// TIA Portal project "chiller" (V19)

(* hardware
DEVICE "S7-1500/ET200MP station_1"  S7-1500 station
   slot 0: "Rail_0"  Rack  6ES7 590-1***0-0AA0
   slot 1: "PLC_1"  CPU 1513-1 PN  6ES7 513-1AM03-0AB0  V3.1
      slot 3: "CPU display_1"  6ES7591-1AA00-0AA0
      slot 32768: "PROFINET interface_1"  X1
         slot 32769: "Port_1"  X1 P1
         slot 32770: "Port_2"  X1 P2
      slot 34817: "Virtual CP interface port_1"  Virtual CP interface port  Virtual CP interface port
   slot 2: "DI 16x24VDC BA_1"  DI 16x24VDC BA  6ES7 521-1BH10-0AA0  V1.1
   slot 3: "DI 16x24VDC BA_2"  DI 16x24VDC BA  6ES7 521-1BH10-0AA0  V1.1
   slot 4: "DQ 16x24VDC/0.5A BA_1"  DQ 16x24VDC/0.5A BA  6ES7 522-1BH10-0AA0  V1.1
   slot 5: "AI 16xI BA_1"  AI 16xI BA  6ES7 531-7MH00-0AB0  V1.0
   slot 6: "AQ 8xU/I HS_1"  AQ 8xU/I HS  6ES7 532-5HF00-0AB0  V2.2
DEVICE "HMI_1"  TP700 Comfort
   slot 0: "HMI_1"  TP700 Comfort  6AV2 124-0GC01-0AX0  17.0.0.0
   slot 1: "HMI_RT_1"  TP700 Comfort  6AV2 124-0GC01-0AX0  17.0.0.0
   slot 5: "HMI_1.IE_CP_1"  PROFINET Interface  17.0.0.0
      slot 1: "PROFINET Interface_1"  PROFINET Interface
         slot 1: "Port_1"  Port
         slot 2: "Port_2"  Port
   slot 7: "HMI_1.MPI/DP_CP_1"  MPI/DP Interface  17.0.0.0
*)

// ===== PLC "PLC_1"  CPU 1513-1 PN =====

VAR_GLOBAL   // PLC tag table "IO_Inputs"
   "I0.0" AT %I0.0 : Bool;
   "I0.1" AT %I0.1 : Bool;
   "I0.2" AT %I0.2 : Bool;
   "I0.3" AT %I0.3 : Bool;
   "I0.4" AT %I0.4 : Bool;
   "I0.5" AT %I0.5 : Bool;
   "I0.6" AT %I0.6 : Bool;
   "I0.7" AT %I0.7 : Bool;
   "I1.0" AT %I1.0 : Bool;
   "I1.1" AT %I1.1 : Bool;
   "I1.2" AT %I1.2 : Bool;
   "I1.3" AT %I1.3 : Bool;
   "I1.4" AT %I1.4 : Bool;
   "I1.5" AT %I1.5 : Bool;
   "I1.6" AT %I1.6 : Bool;
   "I1.7" AT %I1.7 : Bool;
   "I_Comp06_OffFb" AT %I2.0 : Bool;
   "I_Comp06_Fault" AT %I2.1 : Bool;
   "I_Comp07_OnFb" AT %I2.2 : Bool;
   "I_Comp07_OffFb" AT %I2.3 : Bool;
   "I_Comp07_Fault" AT %I2.4 : Bool;
   "I_Comp08_OnFb" AT %I2.5 : Bool;
   "I_Comp08_OffFb" AT %I2.6 : Bool;
   "I_Comp08_Fault" AT %I2.7 : Bool;
   "System_Byte" AT %MB1 : Byte;
   "FirstScan" AT %M1.0 : Bool;
   "DiagStatusUpdate" AT %M1.1 : Bool;
   "AlwaysTRUE" AT %M1.2 : Bool;
   "AlwaysFALSE" AT %M1.3 : Bool;
   "Clock_Byte" AT %MB10 : Byte;
   "Clock_10Hz" AT %M10.0 : Bool;
   "Clock_5Hz" AT %M10.1 : Bool;
   "Clock_2.5Hz" AT %M10.2 : Bool;
   "Clock_2Hz" AT %M10.3 : Bool;
   "Clock_1.25Hz" AT %M10.4 : Bool;
   "Clock_1Hz" AT %M10.5 : Bool;
   "Clock_0.625Hz" AT %M10.6 : Bool;
   "Clock_0.5Hz" AT %M10.7 : Bool;
   "Tag_1" AT %I34.0 : Bool;
END_VAR

VAR_GLOBAL   // PLC tag table "IO_Outputs"
   "Q_Comp01_Start" AT %I3.0 : Bool;
   "Q_Comp02_Start" AT %I3.1 : Bool;
   "Q_Comp03_Start" AT %I3.2 : Bool;
   "Q_Comp04_Start" AT %I3.3 : Bool;
   "Q_Comp05_Start" AT %I3.4 : Bool;
   "Q_Comp06_Start" AT %I3.5 : Bool;
   "Q_Comp07_Start" AT %I3.6 : Bool;
   "Q_Comp08_Start" AT %I3.7 : Bool;
END_VAR

TYPE "UDT_Process"
   STRUCT
      WaterOutletTemp : Real;
      WaterTempSetPoint : Real;
      GasPressure : Real;
      GasPressureSetPoint : Real;
      CompressorDemand : Real;
      FanDemand : Real;
      RunningCompressorCount : Int;
      RunningFanCount : Int;
      CompressorPercent : Real;
      FanPercent : Real;
      RequiredCompressorCount : Int;
      RequestedCompressorCount : Int;
      RequiredFanCount : Int;
      RequestedFanCount : Int;
   END_STRUCT;
END_TYPE

TYPE "UDT_Fan"
   STRUCT
      IO : Struct
         DI_OnFeedback : Bool;
         DI_OffFeedback : Bool;
         DI_Fault : Bool;
         DO_Start : Bool;
      END_STRUCT;
      Cfg : Struct
         Enabled : Bool;
      END_STRUCT;
      Sts : Struct
         Runnig : Bool;
         Ready : Bool;
         Status : Int;
      END_STRUCT;
      Cmd : Struct
         StartRequest : Bool;
         ResetFault : Bool;
      END_STRUCT;
      Flt : Struct
         FeedbackFault : Bool;
         AnyFault : Bool;
      END_STRUCT;
   END_STRUCT;
END_TYPE

TYPE "UDT_Compressor"
   STRUCT
      Cfg : Struct
         Enabled : Bool;
      END_STRUCT;
      Sts : Struct
         Running : Bool;
         Ready : Bool;
         Status : Int;
         RunSeconds : DInt;
         RunHours : Real;
      END_STRUCT;
      Cmd : Struct
         StartRequest : Bool;
         ResetFault : Bool;
         ResetRuntime : Bool;
      END_STRUCT;
      Flt : Struct
         FeedbackFault : Bool;
         AnyFault : Bool;
      END_STRUCT;
      IO : Struct
         DI_OnFeedback : Bool;
         DI_OffFeedback : Bool;
         DI_Fault : Bool;
         DO_Start : Bool;
      END_STRUCT;
   END_STRUCT;
END_TYPE

TYPE "UDT_TimingParams"
   STRUCT
      MinOffTime : Time;
      MinOnTime : Time;
      FeedbackTime : Time;
   END_STRUCT;
END_TYPE

// folder: 00_main

DATA_BLOCK "DB_EquipmentMain"   // DB3
{ S7_Optimized_Access := 'TRUE' }
VERSION : 0.1
// stored: InstanceOfName FB_EquipmentMain
"FB_EquipmentMain"
BEGIN
END_DATA_BLOCK

DATA_BLOCK "DB_MachineMain"   // DB5
{ S7_Optimized_Access := 'TRUE' }
VERSION : 0.1
// stored: InstanceOfName FB_MachineMain
"FB_MachineMain"
BEGIN
END_DATA_BLOCK

DATA_BLOCK "DB_SimulationMain"   // DB6
{ S7_Optimized_Access := 'TRUE' }
VERSION : 0.1
// stored: InstanceOfName FB_SimulationMain
"FB_SimulationMain"
BEGIN
END_DATA_BLOCK

// folder: 03_globalData

DATA_BLOCK "Db_Equipment"   // DB1
{ S7_Optimized_Access := 'TRUE' }
VERSION : 0.1
   VAR
      Compressor : Array[1..8] of "UDT_Compressor";
      Process : "UDT_Process";
      Fan : Array[1..12] of "UDT_Fan";
      CompressorTiming : "UDT_TimingParams";
      FanTiming : "UDT_TimingParams";
   END_VAR
BEGIN
END_DATA_BLOCK

DATA_BLOCK "DB_Machine"   // DB2
{ S7_Optimized_Access := 'TRUE' }
VERSION : 0.1
   VAR
      AutoMode : Bool;
      ManualMode : Bool;
      StartRequest : Bool;
      StopRequest : Bool;
      Running : Bool;
      Ready : Bool;
      AnyFault : Bool;
      DisableAllEquipment : Bool;
      EnableAllEquipment : Bool;
      ResetAllEquipmentFaults : Bool;
      WaterFlowOK : Bool;
      LowTempFault : Bool;
      LowTempLimit : Real;
      WaterFlowFaultDelay : Time;
      LowTempFaultDelay : Time;
      WaterFlowFault : Bool;
   END_VAR
BEGIN
END_DATA_BLOCK

DATA_BLOCK "DB_Simulation"   // DB4
{ S7_Optimized_Access := 'TRUE' }
VERSION : 0.1
   VAR
      Enabled : Bool;
      CompressorOnFb : Array[1..8] of Bool;
      CompressorOffFb : Array[1..8] of Bool;
      CompressorFault : Array[1..8] of Bool;
      FanOnFb : Array[1..12] of Bool;
      FanOffFb : Array[1..12] of Bool;
      FanFaultFb : Array[1..12] of Bool;
   END_VAR
BEGIN
END_DATA_BLOCK

DATA_BLOCK "DB_Alarm"   // DB9
{ S7_Optimized_Access := 'TRUE' }
VERSION : 0.1
   VAR
      AlarmWord1 : Word;
      AlarmWord2 : Word;
   END_VAR
BEGIN
END_DATA_BLOCK

// folder: 00_main

FUNCTION_BLOCK "FB_MachineMain"   // FB5, LAD
{ S7_Optimized_Access := 'TRUE' }
VERSION : 0.1
   VAR
      tWaterFlowFault : TON_TIME;
      tLowTempFault : TON_TIME;
   END_VAR
   VAR_TEMP
      WaterFlowTimeout : Bool;
      LowTempTimeout : Bool;
   END_VAR
BEGIN

REGION Network 1
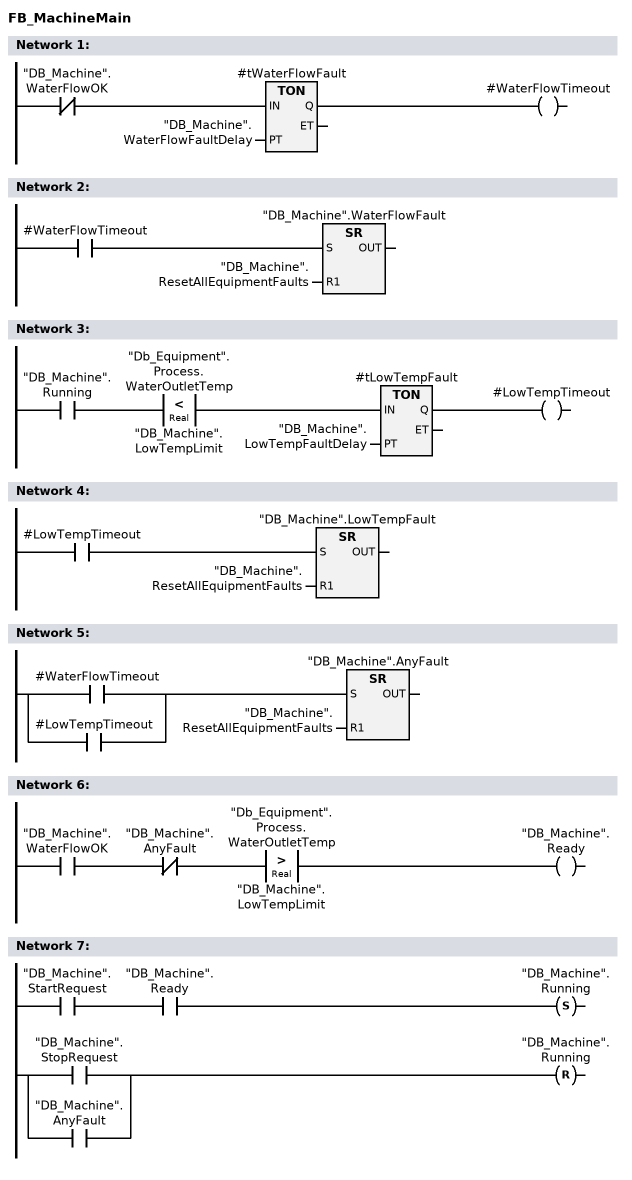
   #tWaterFlowFault(IN := NOT "DB_Machine".WaterFlowOK, PT := "DB_Machine".WaterFlowFaultDelay);   // TON
   #WaterFlowTimeout := #tWaterFlowFault.Q;
END_REGION

REGION Network 2
   RUNG wire#powerrail
      Contact( #WaterFlowTimeout )
      S_SR(operand := "DB_Machine".WaterFlowFault, r1 := "DB_Machine".ResetAllEquipmentFaults)
   END_RUNG
   // the same network as SCL:
   IF #WaterFlowTimeout THEN
       "DB_Machine".WaterFlowFault := TRUE;   // SR flip-flop
   END_IF;
   IF "DB_Machine".ResetAllEquipmentFaults THEN "DB_Machine".WaterFlowFault := FALSE; END_IF;
END_REGION

REGION Network 3
   #tLowTempFault(IN := "DB_Machine".Running AND ("Db_Equipment".Process.WaterOutletTemp < "DB_Machine".LowTempLimit),   // TON
                  PT := "DB_Machine".LowTempFaultDelay);
   #LowTempTimeout := #tLowTempFault.Q;
END_REGION

REGION Network 4
   RUNG wire#powerrail
      Contact( #LowTempTimeout )
      S_SR(operand := "DB_Machine".LowTempFault, r1 := "DB_Machine".ResetAllEquipmentFaults)
   END_RUNG
   // the same network as SCL:
   IF #LowTempTimeout THEN
       "DB_Machine".LowTempFault := TRUE;   // SR flip-flop
   END_IF;
   IF "DB_Machine".ResetAllEquipmentFaults THEN "DB_Machine".LowTempFault := FALSE; END_IF;
END_REGION

REGION Network 5
   RUNG wire#powerrail
      Contact( #WaterFlowTimeout )
      wire#w1
      S_SR(operand := "DB_Machine".AnyFault, r1 := "DB_Machine".ResetAllEquipmentFaults)
   END_RUNG
   RUNG wire#powerrail
      Contact( #LowTempTimeout )
   END_RUNG wire#w1
   // the same network as SCL:
   IF #WaterFlowTimeout OR #LowTempTimeout THEN
       "DB_Machine".AnyFault := TRUE;   // SR flip-flop
   END_IF;
   IF "DB_Machine".ResetAllEquipmentFaults THEN "DB_Machine".AnyFault := FALSE; END_IF;
END_REGION

REGION Network 6
   RUNG wire#powerrail
      Contact( "DB_Machine".WaterFlowOK )
      I_Contact( "DB_Machine".AnyFault )
      { S7_Templates := "SrcType := Real" } GT_Contact(in1 := "Db_Equipment".Process.WaterOutletTemp, in2 := "DB_Machine".LowTempLimit)
      Coil( "DB_Machine".Ready )
   END_RUNG
   // the same network as SCL:
   "DB_Machine".Ready := "DB_Machine".WaterFlowOK AND NOT "DB_Machine".AnyFault AND ("Db_Equipment".Process.WaterOutletTemp > "DB_Machine".LowTempLimit);
END_REGION

REGION Network 7
   RUNG wire#powerrail
      Contact( "DB_Machine".StartRequest )
      Contact( "DB_Machine".Ready )
      S_Coil( "DB_Machine".Running )
   END_RUNG
   RUNG wire#powerrail
      Contact( "DB_Machine".StopRequest )
      wire#w1
      R_Coil( "DB_Machine".Running )
   END_RUNG
   RUNG wire#powerrail
      Contact( "DB_Machine".AnyFault )
   END_RUNG wire#w1
   // the same network as SCL:
   IF "DB_Machine".StartRequest AND "DB_Machine".Ready THEN "DB_Machine".Running := TRUE; END_IF;
   IF "DB_Machine".StopRequest OR "DB_Machine".AnyFault THEN "DB_Machine".Running := FALSE; END_IF;
END_REGION
END_FUNCTION_BLOCK

FUNCTION_BLOCK "FB_EquipmentMain"   // FB6, LAD
{ S7_Optimized_Access := 'TRUE' }
VERSION : 0.1
   VAR
      Comp01 : "FB_Compressor";
      Comp02 : "FB_Compressor";
      Comp03 : "FB_Compressor";
      Comp04 : "FB_Compressor";
      Comp05 : "FB_Compressor";
      Comp06 : "FB_Compressor";
      Comp07 : "FB_Compressor";
      Comp08 : "FB_Compressor";
      Comp09 : "FB_Compressor";
      FB_CompressorManager : "FB_CompressorManager";
      Fan01 : "FB_Fan";
      Fan02 : "FB_Fan";
      Fan03 : "FB_Fan";
      Fan04 : "FB_Fan";
      Fan05 : "FB_Fan";
      Fan06 : "FB_Fan";
      Fan07 : "FB_Fan";
      Fan08 : "FB_Fan";
      Fan09 : "FB_Fan";
      Fan10 : "FB_Fan";
      Fan11 : "FB_Fan";
      Fan12 : "FB_Fan";
      FanManager : "FB_FanManager";
   END_VAR
   VAR_TEMP
      FanControlEnable : Bool;
   END_VAR
BEGIN

REGION Network 1
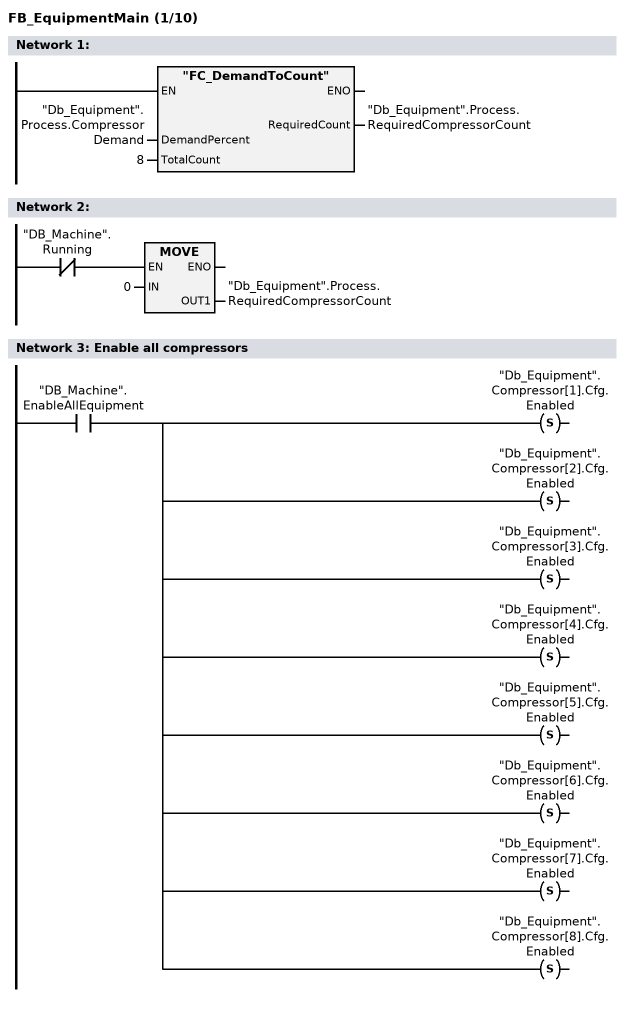
   RUNG wire#powerrail
      "FC_DemandToCount"(DemandPercent := "Db_Equipment".Process.CompressorDemand, TotalCount := 8, RequiredCount => "Db_Equipment".Process.RequiredCompressorCount)
   END_RUNG
   // the same network as SCL:
   "FC_DemandToCount"(DemandPercent := "Db_Equipment".Process.CompressorDemand,
                      TotalCount := 8,
                      RequiredCount => "Db_Equipment".Process.RequiredCompressorCount);
END_REGION

REGION Network 2
   RUNG wire#powerrail
      I_Contact( "DB_Machine".Running )
      Move(in := 0, out1 => "Db_Equipment".Process.RequiredCompressorCount)
   END_RUNG
   // the same network as SCL:
   IF NOT "DB_Machine".Running THEN "Db_Equipment".Process.RequiredCompressorCount := 0; END_IF;
END_REGION

REGION Network 3: Enable all compressors
   RUNG wire#powerrail
      Contact( "DB_Machine".EnableAllEquipment )
      wire#w1
      S_Coil( "Db_Equipment".Compressor[1].Cfg.Enabled )
   END_RUNG
   RUNG wire#w1
      S_Coil( "Db_Equipment".Compressor[2].Cfg.Enabled )
   END_RUNG
   RUNG wire#w1
      S_Coil( "Db_Equipment".Compressor[3].Cfg.Enabled )
   END_RUNG
   RUNG wire#w1
      S_Coil( "Db_Equipment".Compressor[4].Cfg.Enabled )
   END_RUNG
   RUNG wire#w1
      S_Coil( "Db_Equipment".Compressor[5].Cfg.Enabled )
   END_RUNG
   RUNG wire#w1
      S_Coil( "Db_Equipment".Compressor[6].Cfg.Enabled )
   END_RUNG
   RUNG wire#w1
      S_Coil( "Db_Equipment".Compressor[7].Cfg.Enabled )
   END_RUNG
   RUNG wire#w1
      S_Coil( "Db_Equipment".Compressor[8].Cfg.Enabled )
   END_RUNG
   // the same network as SCL:
   IF "DB_Machine".EnableAllEquipment THEN
       "Db_Equipment".Compressor[1].Cfg.Enabled := TRUE;
       "Db_Equipment".Compressor[2].Cfg.Enabled := TRUE;
       "Db_Equipment".Compressor[3].Cfg.Enabled := TRUE;
       "Db_Equipment".Compressor[4].Cfg.Enabled := TRUE;
       "Db_Equipment".Compressor[5].Cfg.Enabled := TRUE;
       "Db_Equipment".Compressor[6].Cfg.Enabled := TRUE;
       "Db_Equipment".Compressor[7].Cfg.Enabled := TRUE;
       "Db_Equipment".Compressor[8].Cfg.Enabled := TRUE;
   END_IF;
END_REGION

REGION Network 4: Enable all fans
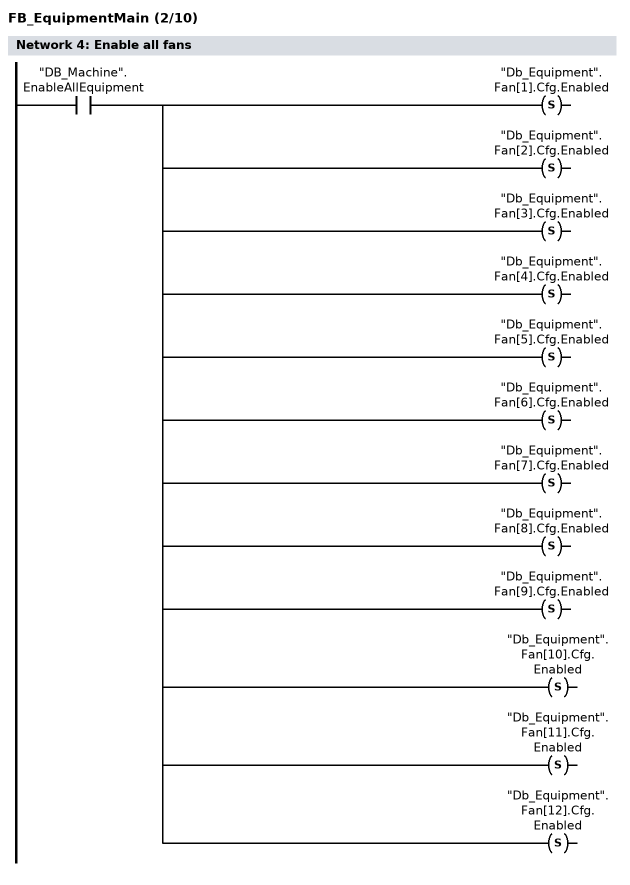
   RUNG wire#powerrail
      Contact( "DB_Machine".EnableAllEquipment )
      wire#w1
      S_Coil( "Db_Equipment".Fan[1].Cfg.Enabled )
   END_RUNG
   RUNG wire#w1
      S_Coil( "Db_Equipment".Fan[2].Cfg.Enabled )
   END_RUNG
   RUNG wire#w1
      S_Coil( "Db_Equipment".Fan[3].Cfg.Enabled )
   END_RUNG
   RUNG wire#w1
      S_Coil( "Db_Equipment".Fan[4].Cfg.Enabled )
   END_RUNG
   RUNG wire#w1
      S_Coil( "Db_Equipment".Fan[5].Cfg.Enabled )
   END_RUNG
   RUNG wire#w1
      S_Coil( "Db_Equipment".Fan[6].Cfg.Enabled )
   END_RUNG
   RUNG wire#w1
      S_Coil( "Db_Equipment".Fan[7].Cfg.Enabled )
   END_RUNG
   RUNG wire#w1
      S_Coil( "Db_Equipment".Fan[8].Cfg.Enabled )
   END_RUNG
   RUNG wire#w1
      S_Coil( "Db_Equipment".Fan[9].Cfg.Enabled )
   END_RUNG
   RUNG wire#w1
      S_Coil( "Db_Equipment".Fan[10].Cfg.Enabled )
   END_RUNG
   RUNG wire#w1
      S_Coil( "Db_Equipment".Fan[11].Cfg.Enabled )
   END_RUNG
   RUNG wire#w1
      S_Coil( "Db_Equipment".Fan[12].Cfg.Enabled )
   END_RUNG
   // the same network as SCL:
   IF "DB_Machine".EnableAllEquipment THEN
       "Db_Equipment".Fan[1].Cfg.Enabled := TRUE;
       "Db_Equipment".Fan[2].Cfg.Enabled := TRUE;
       "Db_Equipment".Fan[3].Cfg.Enabled := TRUE;
       "Db_Equipment".Fan[4].Cfg.Enabled := TRUE;
       "Db_Equipment".Fan[5].Cfg.Enabled := TRUE;
       "Db_Equipment".Fan[6].Cfg.Enabled := TRUE;
       "Db_Equipment".Fan[7].Cfg.Enabled := TRUE;
       "Db_Equipment".Fan[8].Cfg.Enabled := TRUE;
       "Db_Equipment".Fan[9].Cfg.Enabled := TRUE;
       "Db_Equipment".Fan[10].Cfg.Enabled := TRUE;
       "Db_Equipment".Fan[11].Cfg.Enabled := TRUE;
       "Db_Equipment".Fan[12].Cfg.Enabled := TRUE;
   END_IF;
END_REGION

REGION Network 5
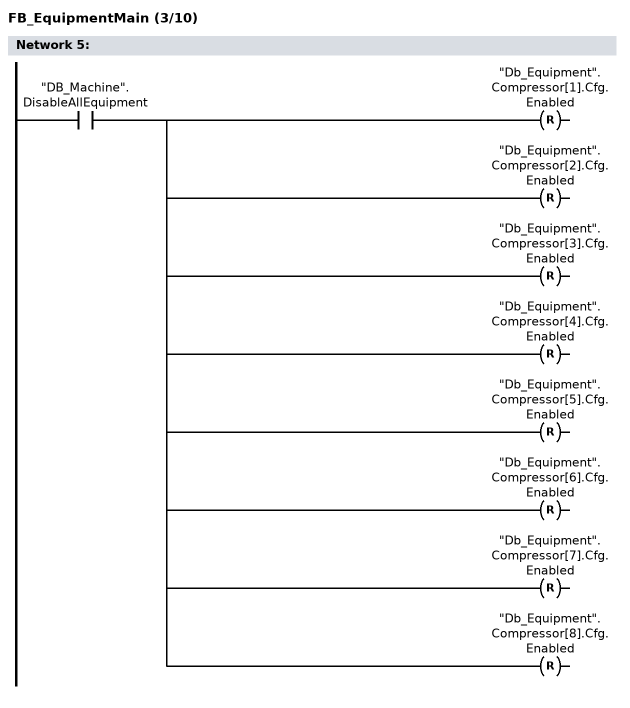
   RUNG wire#powerrail
      Contact( "DB_Machine".DisableAllEquipment )
      wire#w1
      R_Coil( "Db_Equipment".Compressor[1].Cfg.Enabled )
   END_RUNG
   RUNG wire#w1
      R_Coil( "Db_Equipment".Compressor[2].Cfg.Enabled )
   END_RUNG
   RUNG wire#w1
      R_Coil( "Db_Equipment".Compressor[3].Cfg.Enabled )
   END_RUNG
   RUNG wire#w1
      R_Coil( "Db_Equipment".Compressor[4].Cfg.Enabled )
   END_RUNG
   RUNG wire#w1
      R_Coil( "Db_Equipment".Compressor[5].Cfg.Enabled )
   END_RUNG
   RUNG wire#w1
      R_Coil( "Db_Equipment".Compressor[6].Cfg.Enabled )
   END_RUNG
   RUNG wire#w1
      R_Coil( "Db_Equipment".Compressor[7].Cfg.Enabled )
   END_RUNG
   RUNG wire#w1
      R_Coil( "Db_Equipment".Compressor[8].Cfg.Enabled )
   END_RUNG
   // the same network as SCL:
   IF "DB_Machine".DisableAllEquipment THEN
       "Db_Equipment".Compressor[1].Cfg.Enabled := FALSE;
       "Db_Equipment".Compressor[2].Cfg.Enabled := FALSE;
       "Db_Equipment".Compressor[3].Cfg.Enabled := FALSE;
       "Db_Equipment".Compressor[4].Cfg.Enabled := FALSE;
       "Db_Equipment".Compressor[5].Cfg.Enabled := FALSE;
       "Db_Equipment".Compressor[6].Cfg.Enabled := FALSE;
       "Db_Equipment".Compressor[7].Cfg.Enabled := FALSE;
       "Db_Equipment".Compressor[8].Cfg.Enabled := FALSE;
   END_IF;
END_REGION

REGION Network 6
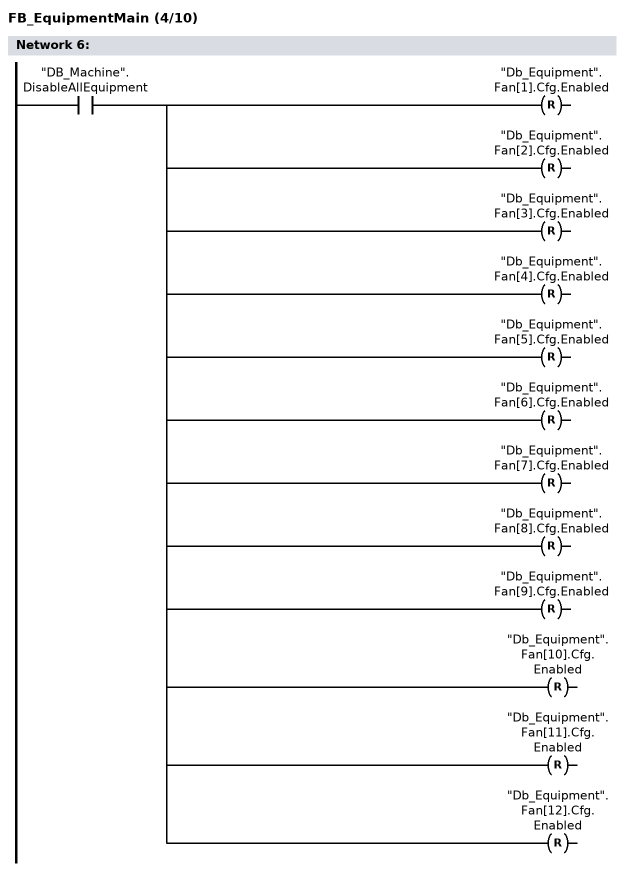
   RUNG wire#powerrail
      Contact( "DB_Machine".DisableAllEquipment )
      wire#w1
      R_Coil( "Db_Equipment".Fan[1].Cfg.Enabled )
   END_RUNG
   RUNG wire#w1
      R_Coil( "Db_Equipment".Fan[2].Cfg.Enabled )
   END_RUNG
   RUNG wire#w1
      R_Coil( "Db_Equipment".Fan[3].Cfg.Enabled )
   END_RUNG
   RUNG wire#w1
      R_Coil( "Db_Equipment".Fan[4].Cfg.Enabled )
   END_RUNG
   RUNG wire#w1
      R_Coil( "Db_Equipment".Fan[5].Cfg.Enabled )
   END_RUNG
   RUNG wire#w1
      R_Coil( "Db_Equipment".Fan[6].Cfg.Enabled )
   END_RUNG
   RUNG wire#w1
      R_Coil( "Db_Equipment".Fan[7].Cfg.Enabled )
   END_RUNG
   RUNG wire#w1
      R_Coil( "Db_Equipment".Fan[8].Cfg.Enabled )
   END_RUNG
   RUNG wire#w1
      R_Coil( "Db_Equipment".Fan[9].Cfg.Enabled )
   END_RUNG
   RUNG wire#w1
      R_Coil( "Db_Equipment".Fan[10].Cfg.Enabled )
   END_RUNG
   RUNG wire#w1
      R_Coil( "Db_Equipment".Fan[11].Cfg.Enabled )
   END_RUNG
   RUNG wire#w1
      R_Coil( "Db_Equipment".Fan[12].Cfg.Enabled )
   END_RUNG
   // the same network as SCL:
   IF "DB_Machine".DisableAllEquipment THEN
       "Db_Equipment".Fan[1].Cfg.Enabled := FALSE;
       "Db_Equipment".Fan[2].Cfg.Enabled := FALSE;
       "Db_Equipment".Fan[3].Cfg.Enabled := FALSE;
       "Db_Equipment".Fan[4].Cfg.Enabled := FALSE;
       "Db_Equipment".Fan[5].Cfg.Enabled := FALSE;
       "Db_Equipment".Fan[6].Cfg.Enabled := FALSE;
       "Db_Equipment".Fan[7].Cfg.Enabled := FALSE;
       "Db_Equipment".Fan[8].Cfg.Enabled := FALSE;
       "Db_Equipment".Fan[9].Cfg.Enabled := FALSE;
       "Db_Equipment".Fan[10].Cfg.Enabled := FALSE;
       "Db_Equipment".Fan[11].Cfg.Enabled := FALSE;
       "Db_Equipment".Fan[12].Cfg.Enabled := FALSE;
   END_IF;
END_REGION

REGION Network 7: Reset compressor faults
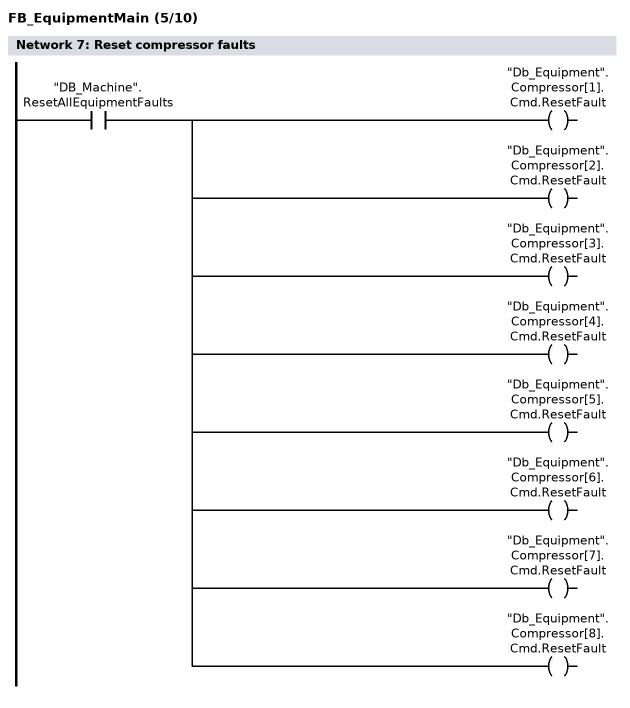
   RUNG wire#powerrail
      Contact( "DB_Machine".ResetAllEquipmentFaults )
      wire#w1
      Coil( "Db_Equipment".Compressor[1].Cmd.ResetFault )
   END_RUNG
   RUNG wire#w1
      Coil( "Db_Equipment".Compressor[2].Cmd.ResetFault )
   END_RUNG
   RUNG wire#w1
      Coil( "Db_Equipment".Compressor[3].Cmd.ResetFault )
   END_RUNG
   RUNG wire#w1
      Coil( "Db_Equipment".Compressor[4].Cmd.ResetFault )
   END_RUNG
   RUNG wire#w1
      Coil( "Db_Equipment".Compressor[5].Cmd.ResetFault )
   END_RUNG
   RUNG wire#w1
      Coil( "Db_Equipment".Compressor[6].Cmd.ResetFault )
   END_RUNG
   RUNG wire#w1
      Coil( "Db_Equipment".Compressor[7].Cmd.ResetFault )
   END_RUNG
   RUNG wire#w1
      Coil( "Db_Equipment".Compressor[8].Cmd.ResetFault )
   END_RUNG
   // the same network as SCL:
   "Db_Equipment".Compressor[1].Cmd.ResetFault := "DB_Machine".ResetAllEquipmentFaults;
   "Db_Equipment".Compressor[2].Cmd.ResetFault := "DB_Machine".ResetAllEquipmentFaults;
   "Db_Equipment".Compressor[3].Cmd.ResetFault := "DB_Machine".ResetAllEquipmentFaults;
   "Db_Equipment".Compressor[4].Cmd.ResetFault := "DB_Machine".ResetAllEquipmentFaults;
   "Db_Equipment".Compressor[5].Cmd.ResetFault := "DB_Machine".ResetAllEquipmentFaults;
   "Db_Equipment".Compressor[6].Cmd.ResetFault := "DB_Machine".ResetAllEquipmentFaults;
   "Db_Equipment".Compressor[7].Cmd.ResetFault := "DB_Machine".ResetAllEquipmentFaults;
   "Db_Equipment".Compressor[8].Cmd.ResetFault := "DB_Machine".ResetAllEquipmentFaults;
END_REGION

REGION Network 8: Reset fan faults
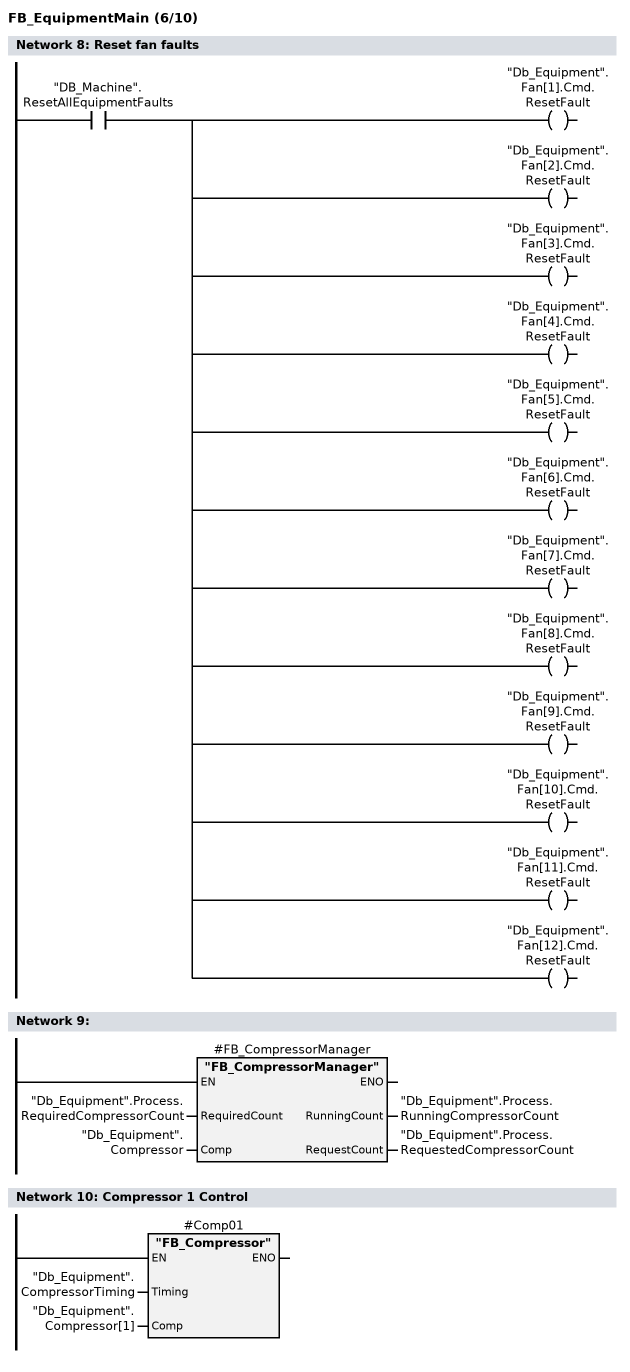
   RUNG wire#powerrail
      Contact( "DB_Machine".ResetAllEquipmentFaults )
      wire#w1
      Coil( "Db_Equipment".Fan[1].Cmd.ResetFault )
   END_RUNG
   RUNG wire#w1
      Coil( "Db_Equipment".Fan[2].Cmd.ResetFault )
   END_RUNG
   RUNG wire#w1
      Coil( "Db_Equipment".Fan[3].Cmd.ResetFault )
   END_RUNG
   RUNG wire#w1
      Coil( "Db_Equipment".Fan[4].Cmd.ResetFault )
   END_RUNG
   RUNG wire#w1
      Coil( "Db_Equipment".Fan[5].Cmd.ResetFault )
   END_RUNG
   RUNG wire#w1
      Coil( "Db_Equipment".Fan[6].Cmd.ResetFault )
   END_RUNG
   RUNG wire#w1
      Coil( "Db_Equipment".Fan[7].Cmd.ResetFault )
   END_RUNG
   RUNG wire#w1
      Coil( "Db_Equipment".Fan[8].Cmd.ResetFault )
   END_RUNG
   RUNG wire#w1
      Coil( "Db_Equipment".Fan[9].Cmd.ResetFault )
   END_RUNG
   RUNG wire#w1
      Coil( "Db_Equipment".Fan[10].Cmd.ResetFault )
   END_RUNG
   RUNG wire#w1
      Coil( "Db_Equipment".Fan[11].Cmd.ResetFault )
   END_RUNG
   RUNG wire#w1
      Coil( "Db_Equipment".Fan[12].Cmd.ResetFault )
   END_RUNG
   // the same network as SCL:
   "Db_Equipment".Fan[1].Cmd.ResetFault := "DB_Machine".ResetAllEquipmentFaults;
   "Db_Equipment".Fan[2].Cmd.ResetFault := "DB_Machine".ResetAllEquipmentFaults;
   "Db_Equipment".Fan[3].Cmd.ResetFault := "DB_Machine".ResetAllEquipmentFaults;
   "Db_Equipment".Fan[4].Cmd.ResetFault := "DB_Machine".ResetAllEquipmentFaults;
   "Db_Equipment".Fan[5].Cmd.ResetFault := "DB_Machine".ResetAllEquipmentFaults;
   "Db_Equipment".Fan[6].Cmd.ResetFault := "DB_Machine".ResetAllEquipmentFaults;
   "Db_Equipment".Fan[7].Cmd.ResetFault := "DB_Machine".ResetAllEquipmentFaults;
   "Db_Equipment".Fan[8].Cmd.ResetFault := "DB_Machine".ResetAllEquipmentFaults;
   "Db_Equipment".Fan[9].Cmd.ResetFault := "DB_Machine".ResetAllEquipmentFaults;
   "Db_Equipment".Fan[10].Cmd.ResetFault := "DB_Machine".ResetAllEquipmentFaults;
   "Db_Equipment".Fan[11].Cmd.ResetFault := "DB_Machine".ResetAllEquipmentFaults;
   "Db_Equipment".Fan[12].Cmd.ResetFault := "DB_Machine".ResetAllEquipmentFaults;
END_REGION

REGION Network 9
   RUNG wire#powerrail
      #FB_CompressorManager(RequiredCount := "Db_Equipment".Process.RequiredCompressorCount, Comp := "Db_Equipment".Compressor, RunningCount => "Db_Equipment".Process.RunningCompressorCount, RequestCount => "Db_Equipment".Process.RequestedCompressorCount)
   END_RUNG
   // the same network as SCL:
   #FB_CompressorManager(RequiredCount := "Db_Equipment".Process.RequiredCompressorCount,   // "FB_CompressorManager"
                         Comp := "Db_Equipment".Compressor,
                         RunningCount => "Db_Equipment".Process.RunningCompressorCount,
                         RequestCount => "Db_Equipment".Process.RequestedCompressorCount);
END_REGION

REGION Network 10: Compressor 1 Control
   RUNG wire#powerrail
      #Comp01(Timing := "Db_Equipment".CompressorTiming, Comp := "Db_Equipment".Compressor[1])
   END_RUNG
   // the same network as SCL:
   #Comp01(Timing := "Db_Equipment".CompressorTiming, Comp := "Db_Equipment".Compressor[1]);   // "FB_Compressor"
END_REGION

REGION Network 11
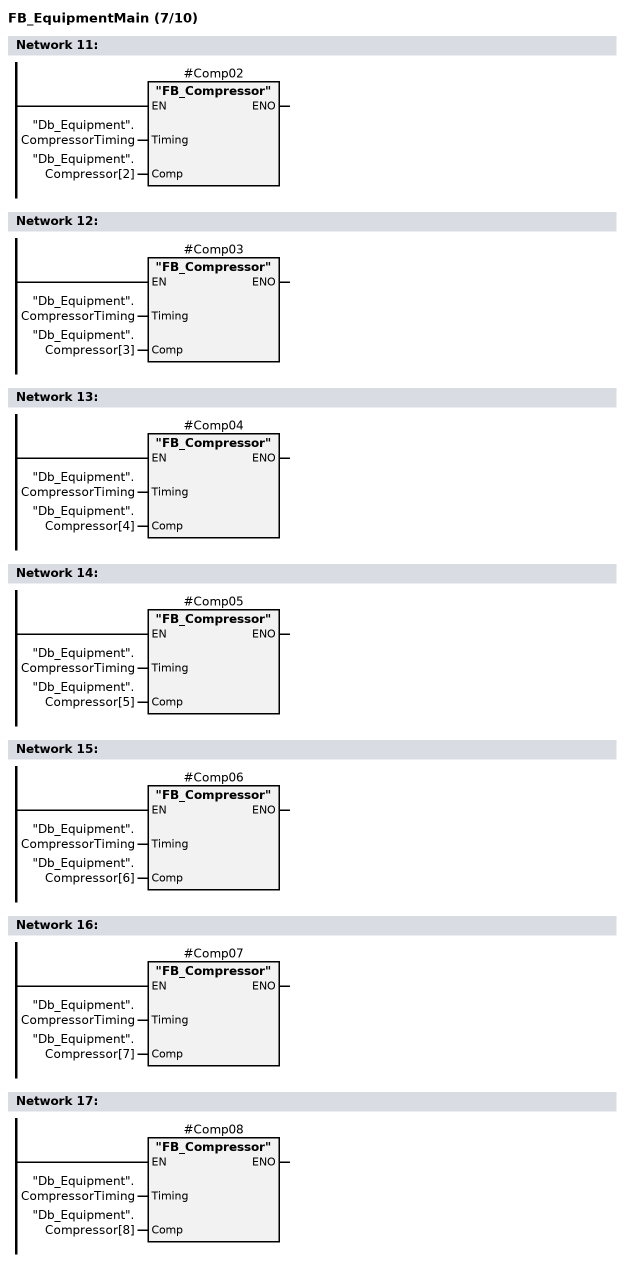
   RUNG wire#powerrail
      #Comp02(Timing := "Db_Equipment".CompressorTiming, Comp := "Db_Equipment".Compressor[2])
   END_RUNG
   // the same network as SCL:
   #Comp02(Timing := "Db_Equipment".CompressorTiming, Comp := "Db_Equipment".Compressor[2]);   // "FB_Compressor"
END_REGION

REGION Network 12
   RUNG wire#powerrail
      #Comp03(Timing := "Db_Equipment".CompressorTiming, Comp := "Db_Equipment".Compressor[3])
   END_RUNG
   // the same network as SCL:
   #Comp03(Timing := "Db_Equipment".CompressorTiming, Comp := "Db_Equipment".Compressor[3]);   // "FB_Compressor"
END_REGION

REGION Network 13
   RUNG wire#powerrail
      #Comp04(Timing := "Db_Equipment".CompressorTiming, Comp := "Db_Equipment".Compressor[4])
   END_RUNG
   // the same network as SCL:
   #Comp04(Timing := "Db_Equipment".CompressorTiming, Comp := "Db_Equipment".Compressor[4]);   // "FB_Compressor"
END_REGION

REGION Network 14
   RUNG wire#powerrail
      #Comp05(Timing := "Db_Equipment".CompressorTiming, Comp := "Db_Equipment".Compressor[5])
   END_RUNG
   // the same network as SCL:
   #Comp05(Timing := "Db_Equipment".CompressorTiming, Comp := "Db_Equipment".Compressor[5]);   // "FB_Compressor"
END_REGION

REGION Network 15
   RUNG wire#powerrail
      #Comp06(Timing := "Db_Equipment".CompressorTiming, Comp := "Db_Equipment".Compressor[6])
   END_RUNG
   // the same network as SCL:
   #Comp06(Timing := "Db_Equipment".CompressorTiming, Comp := "Db_Equipment".Compressor[6]);   // "FB_Compressor"
END_REGION

REGION Network 16
   RUNG wire#powerrail
      #Comp07(Timing := "Db_Equipment".CompressorTiming, Comp := "Db_Equipment".Compressor[7])
   END_RUNG
   // the same network as SCL:
   #Comp07(Timing := "Db_Equipment".CompressorTiming, Comp := "Db_Equipment".Compressor[7]);   // "FB_Compressor"
END_REGION

REGION Network 17
   RUNG wire#powerrail
      #Comp08(Timing := "Db_Equipment".CompressorTiming, Comp := "Db_Equipment".Compressor[8])
   END_RUNG
   // the same network as SCL:
   #Comp08(Timing := "Db_Equipment".CompressorTiming, Comp := "Db_Equipment".Compressor[8]);   // "FB_Compressor"
END_REGION

REGION Network 18
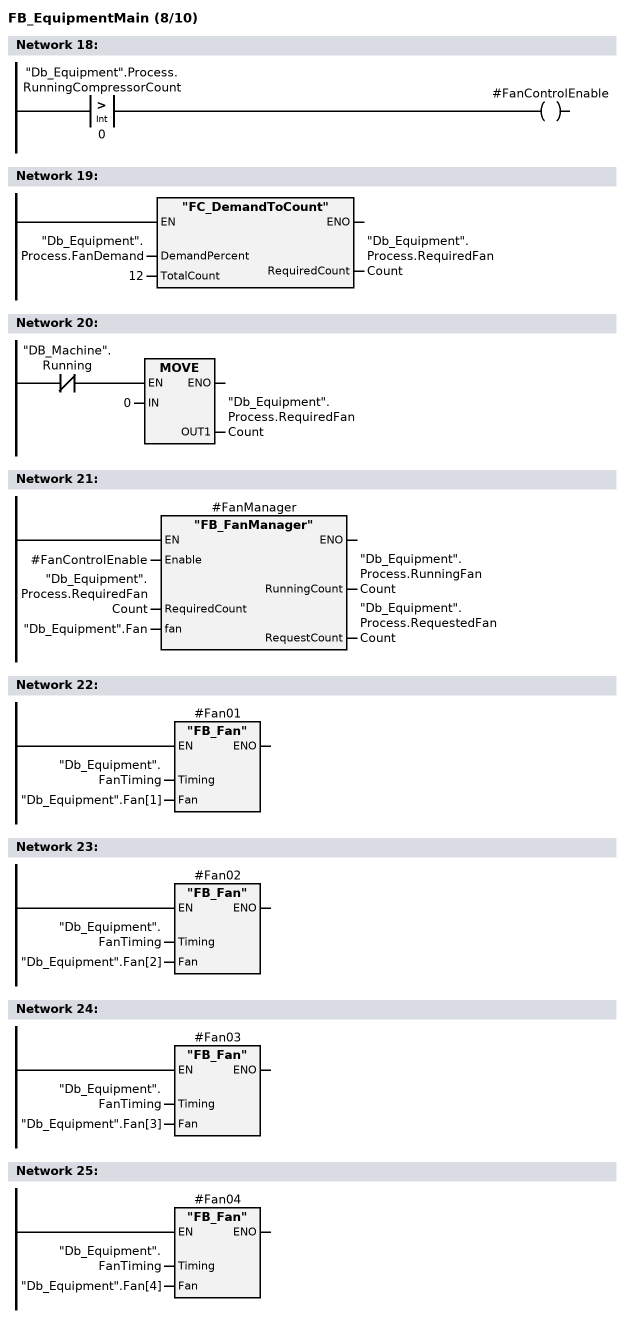
   RUNG wire#powerrail
      { S7_Templates := "SrcType := Int" } GT_Contact(in1 := "Db_Equipment".Process.RunningCompressorCount, in2 := 0)
      Coil( #FanControlEnable )
   END_RUNG
   // the same network as SCL:
   #FanControlEnable := "Db_Equipment".Process.RunningCompressorCount > 0;
END_REGION

REGION Network 19
   RUNG wire#powerrail
      "FC_DemandToCount"(DemandPercent := "Db_Equipment".Process.FanDemand, TotalCount := 12, RequiredCount => "Db_Equipment".Process.RequiredFanCount)
   END_RUNG
   // the same network as SCL:
   "FC_DemandToCount"(DemandPercent := "Db_Equipment".Process.FanDemand,
                      TotalCount := 12,
                      RequiredCount => "Db_Equipment".Process.RequiredFanCount);
END_REGION

REGION Network 20
   RUNG wire#powerrail
      I_Contact( "DB_Machine".Running )
      Move(in := 0, out1 => "Db_Equipment".Process.RequiredFanCount)
   END_RUNG
   // the same network as SCL:
   IF NOT "DB_Machine".Running THEN "Db_Equipment".Process.RequiredFanCount := 0; END_IF;
END_REGION

REGION Network 21
   RUNG wire#powerrail
      #FanManager(Enable := #FanControlEnable, RequiredCount := "Db_Equipment".Process.RequiredFanCount, fan := "Db_Equipment".Fan, RunningCount => "Db_Equipment".Process.RunningFanCount, RequestCount => "Db_Equipment".Process.RequestedFanCount)
   END_RUNG
   // the same network as SCL:
   #FanManager(Enable := #FanControlEnable,   // "FB_FanManager"
               RequiredCount := "Db_Equipment".Process.RequiredFanCount,
               fan := "Db_Equipment".Fan,
               RunningCount => "Db_Equipment".Process.RunningFanCount,
               RequestCount => "Db_Equipment".Process.RequestedFanCount);
END_REGION

REGION Network 22
   RUNG wire#powerrail
      #Fan01(Timing := "Db_Equipment".FanTiming, Fan := "Db_Equipment".Fan[1])
   END_RUNG
   // the same network as SCL:
   #Fan01(Timing := "Db_Equipment".FanTiming, Fan := "Db_Equipment".Fan[1]);   // "FB_Fan"
END_REGION

REGION Network 23
   RUNG wire#powerrail
      #Fan02(Timing := "Db_Equipment".FanTiming, Fan := "Db_Equipment".Fan[2])
   END_RUNG
   // the same network as SCL:
   #Fan02(Timing := "Db_Equipment".FanTiming, Fan := "Db_Equipment".Fan[2]);   // "FB_Fan"
END_REGION

REGION Network 24
   RUNG wire#powerrail
      #Fan03(Timing := "Db_Equipment".FanTiming, Fan := "Db_Equipment".Fan[3])
   END_RUNG
   // the same network as SCL:
   #Fan03(Timing := "Db_Equipment".FanTiming, Fan := "Db_Equipment".Fan[3]);   // "FB_Fan"
END_REGION

REGION Network 25
   RUNG wire#powerrail
      #Fan04(Timing := "Db_Equipment".FanTiming, Fan := "Db_Equipment".Fan[4])
   END_RUNG
   // the same network as SCL:
   #Fan04(Timing := "Db_Equipment".FanTiming, Fan := "Db_Equipment".Fan[4]);   // "FB_Fan"
END_REGION

REGION Network 26
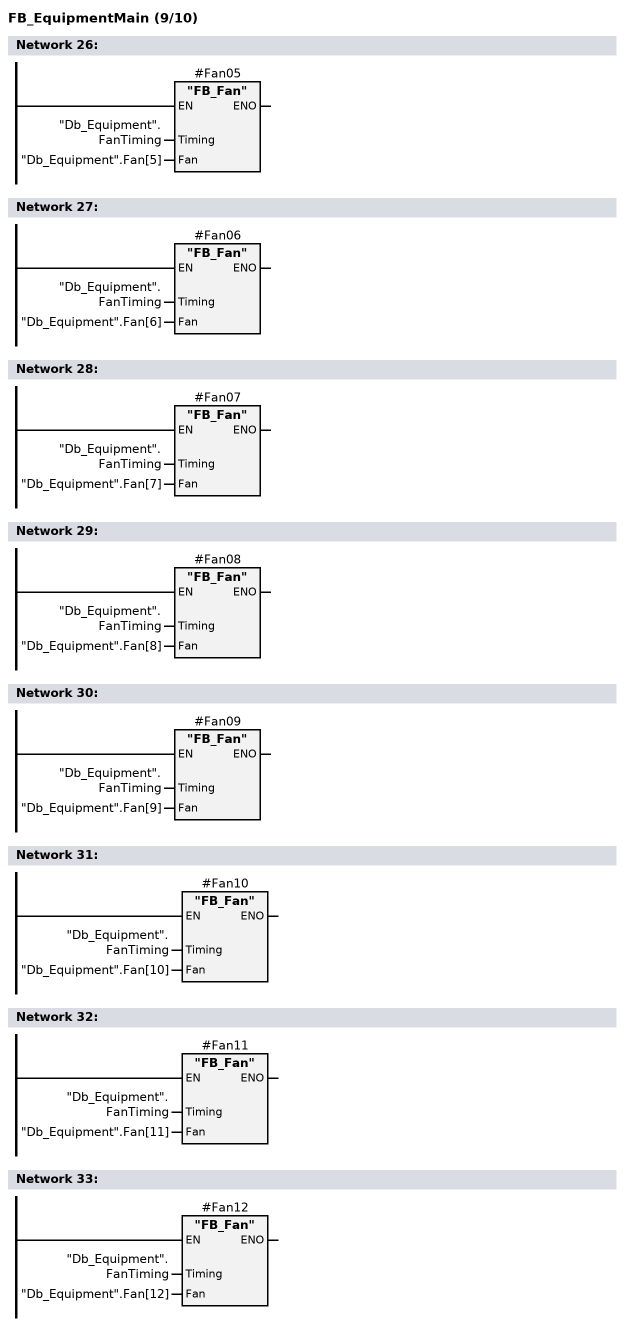
   RUNG wire#powerrail
      #Fan05(Timing := "Db_Equipment".FanTiming, Fan := "Db_Equipment".Fan[5])
   END_RUNG
   // the same network as SCL:
   #Fan05(Timing := "Db_Equipment".FanTiming, Fan := "Db_Equipment".Fan[5]);   // "FB_Fan"
END_REGION

REGION Network 27
   RUNG wire#powerrail
      #Fan06(Timing := "Db_Equipment".FanTiming, Fan := "Db_Equipment".Fan[6])
   END_RUNG
   // the same network as SCL:
   #Fan06(Timing := "Db_Equipment".FanTiming, Fan := "Db_Equipment".Fan[6]);   // "FB_Fan"
END_REGION

REGION Network 28
   RUNG wire#powerrail
      #Fan07(Timing := "Db_Equipment".FanTiming, Fan := "Db_Equipment".Fan[7])
   END_RUNG
   // the same network as SCL:
   #Fan07(Timing := "Db_Equipment".FanTiming, Fan := "Db_Equipment".Fan[7]);   // "FB_Fan"
END_REGION

REGION Network 29
   RUNG wire#powerrail
      #Fan08(Timing := "Db_Equipment".FanTiming, Fan := "Db_Equipment".Fan[8])
   END_RUNG
   // the same network as SCL:
   #Fan08(Timing := "Db_Equipment".FanTiming, Fan := "Db_Equipment".Fan[8]);   // "FB_Fan"
END_REGION

REGION Network 30
   RUNG wire#powerrail
      #Fan09(Timing := "Db_Equipment".FanTiming, Fan := "Db_Equipment".Fan[9])
   END_RUNG
   // the same network as SCL:
   #Fan09(Timing := "Db_Equipment".FanTiming, Fan := "Db_Equipment".Fan[9]);   // "FB_Fan"
END_REGION

REGION Network 31
   RUNG wire#powerrail
      #Fan10(Timing := "Db_Equipment".FanTiming, Fan := "Db_Equipment".Fan[10])
   END_RUNG
   // the same network as SCL:
   #Fan10(Timing := "Db_Equipment".FanTiming, Fan := "Db_Equipment".Fan[10]);   // "FB_Fan"
END_REGION

REGION Network 32
   RUNG wire#powerrail
      #Fan11(Timing := "Db_Equipment".FanTiming, Fan := "Db_Equipment".Fan[11])
   END_RUNG
   // the same network as SCL:
   #Fan11(Timing := "Db_Equipment".FanTiming, Fan := "Db_Equipment".Fan[11]);   // "FB_Fan"
END_REGION

REGION Network 33
   RUNG wire#powerrail
      #Fan12(Timing := "Db_Equipment".FanTiming, Fan := "Db_Equipment".Fan[12])
   END_RUNG
   // the same network as SCL:
   #Fan12(Timing := "Db_Equipment".FanTiming, Fan := "Db_Equipment".Fan[12]);   // "FB_Fan"
END_REGION

REGION Network 34
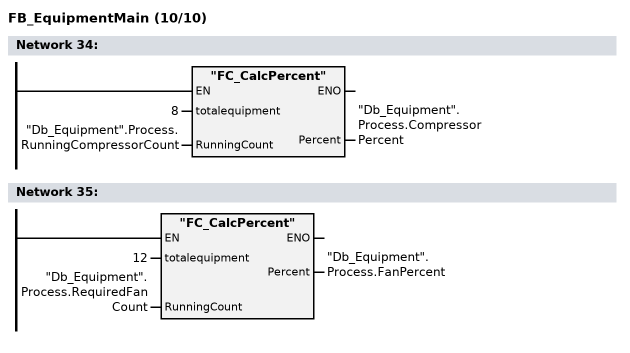
   RUNG wire#powerrail
      "FC_CalcPercent"(totalequipment := 8, RunningCount := "Db_Equipment".Process.RunningCompressorCount, Percent => "Db_Equipment".Process.CompressorPercent)
   END_RUNG
   // the same network as SCL:
   "FC_CalcPercent"(totalequipment := 8,
                    RunningCount := "Db_Equipment".Process.RunningCompressorCount,
                    Percent => "Db_Equipment".Process.CompressorPercent);
END_REGION

REGION Network 35
   RUNG wire#powerrail
      "FC_CalcPercent"(totalequipment := 12, RunningCount := "Db_Equipment".Process.RequiredFanCount, Percent => "Db_Equipment".Process.FanPercent)
   END_RUNG
   // the same network as SCL:
   "FC_CalcPercent"(totalequipment := 12,
                    RunningCount := "Db_Equipment".Process.RequiredFanCount,
                    Percent => "Db_Equipment".Process.FanPercent);
END_REGION
END_FUNCTION_BLOCK

FUNCTION_BLOCK "FB_SimulationMain"   // FB8, LAD
{ S7_Optimized_Access := 'TRUE' }
VERSION : 0.1
   VAR
      Comp08 : "FB_CompressorSim";
      Comp07 : "FB_CompressorSim";
      Comp06 : "FB_CompressorSim";
      Comp05 : "FB_CompressorSim";
      Comp04 : "FB_CompressorSim";
      Comp03 : "FB_CompressorSim";
      Comp02 : "FB_CompressorSim";
      Comp01 : "FB_CompressorSim";
      FanSim01 : "FB_FanSim";
      FanSim02 : "FB_FanSim";
      FanSim03 : "FB_FanSim";
      FanSim04 : "FB_FanSim";
      FanSim05 : "FB_FanSim";
      FanSim06 : "FB_FanSim";
      FanSim07 : "FB_FanSim";
      FanSim08 : "FB_FanSim";
      FanSim09 : "FB_FanSim";
      FanSim10 : "FB_FanSim";
      FanSim11 : "FB_FanSim";
      FanSim12 : "FB_FanSim";
   END_VAR
BEGIN

REGION Network 1
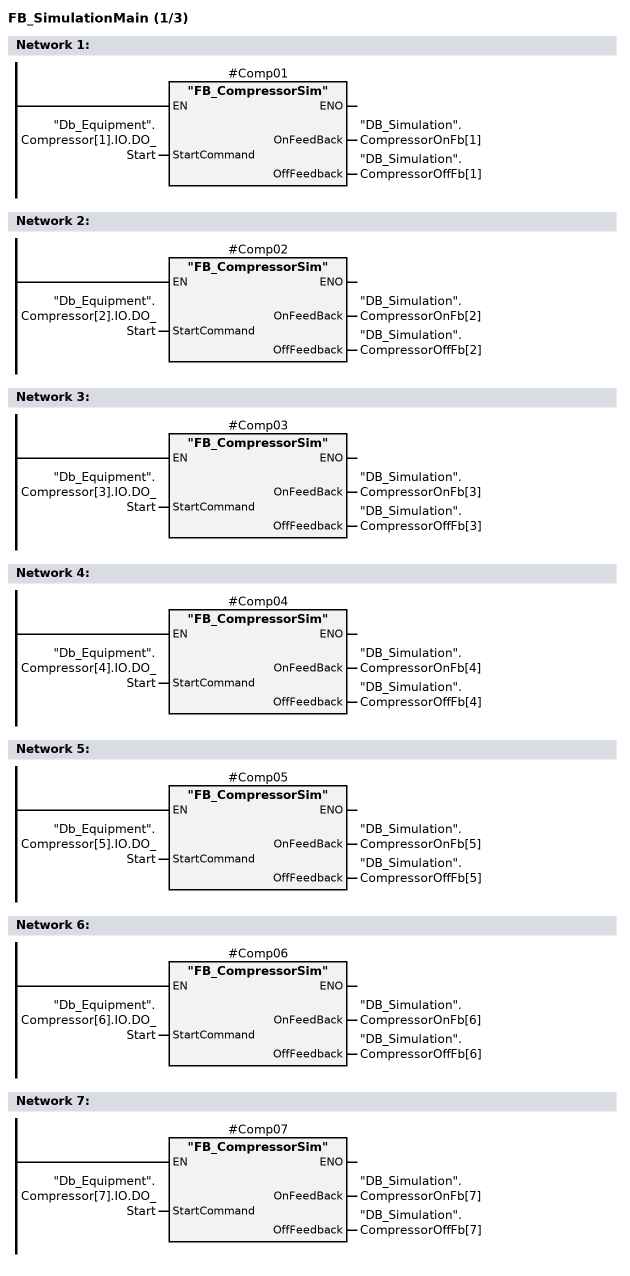
   RUNG wire#powerrail
      #Comp01(StartCommand := "Db_Equipment".Compressor[1].IO.DO_Start, OnFeedBack => "DB_Simulation".CompressorOnFb[1], OffFeedback => "DB_Simulation".CompressorOffFb[1])
   END_RUNG
   // the same network as SCL:
   #Comp01(StartCommand := "Db_Equipment".Compressor[1].IO.DO_Start,   // "FB_CompressorSim"
           OnFeedBack => "DB_Simulation".CompressorOnFb[1],
           OffFeedback => "DB_Simulation".CompressorOffFb[1]);
END_REGION

REGION Network 2
   RUNG wire#powerrail
      #Comp02(StartCommand := "Db_Equipment".Compressor[2].IO.DO_Start, OnFeedBack => "DB_Simulation".CompressorOnFb[2], OffFeedback => "DB_Simulation".CompressorOffFb[2])
   END_RUNG
   // the same network as SCL:
   #Comp02(StartCommand := "Db_Equipment".Compressor[2].IO.DO_Start,   // "FB_CompressorSim"
           OnFeedBack => "DB_Simulation".CompressorOnFb[2],
           OffFeedback => "DB_Simulation".CompressorOffFb[2]);
END_REGION

REGION Network 3
   RUNG wire#powerrail
      #Comp03(StartCommand := "Db_Equipment".Compressor[3].IO.DO_Start, OnFeedBack => "DB_Simulation".CompressorOnFb[3], OffFeedback => "DB_Simulation".CompressorOffFb[3])
   END_RUNG
   // the same network as SCL:
   #Comp03(StartCommand := "Db_Equipment".Compressor[3].IO.DO_Start,   // "FB_CompressorSim"
           OnFeedBack => "DB_Simulation".CompressorOnFb[3],
           OffFeedback => "DB_Simulation".CompressorOffFb[3]);
END_REGION

REGION Network 4
   RUNG wire#powerrail
      #Comp04(StartCommand := "Db_Equipment".Compressor[4].IO.DO_Start, OnFeedBack => "DB_Simulation".CompressorOnFb[4], OffFeedback => "DB_Simulation".CompressorOffFb[4])
   END_RUNG
   // the same network as SCL:
   #Comp04(StartCommand := "Db_Equipment".Compressor[4].IO.DO_Start,   // "FB_CompressorSim"
           OnFeedBack => "DB_Simulation".CompressorOnFb[4],
           OffFeedback => "DB_Simulation".CompressorOffFb[4]);
END_REGION

REGION Network 5
   RUNG wire#powerrail
      #Comp05(StartCommand := "Db_Equipment".Compressor[5].IO.DO_Start, OnFeedBack => "DB_Simulation".CompressorOnFb[5], OffFeedback => "DB_Simulation".CompressorOffFb[5])
   END_RUNG
   // the same network as SCL:
   #Comp05(StartCommand := "Db_Equipment".Compressor[5].IO.DO_Start,   // "FB_CompressorSim"
           OnFeedBack => "DB_Simulation".CompressorOnFb[5],
           OffFeedback => "DB_Simulation".CompressorOffFb[5]);
END_REGION

REGION Network 6
   RUNG wire#powerrail
      #Comp06(StartCommand := "Db_Equipment".Compressor[6].IO.DO_Start, OnFeedBack => "DB_Simulation".CompressorOnFb[6], OffFeedback => "DB_Simulation".CompressorOffFb[6])
   END_RUNG
   // the same network as SCL:
   #Comp06(StartCommand := "Db_Equipment".Compressor[6].IO.DO_Start,   // "FB_CompressorSim"
           OnFeedBack => "DB_Simulation".CompressorOnFb[6],
           OffFeedback => "DB_Simulation".CompressorOffFb[6]);
END_REGION

REGION Network 7
   RUNG wire#powerrail
      #Comp07(StartCommand := "Db_Equipment".Compressor[7].IO.DO_Start, OnFeedBack => "DB_Simulation".CompressorOnFb[7], OffFeedback => "DB_Simulation".CompressorOffFb[7])
   END_RUNG
   // the same network as SCL:
   #Comp07(StartCommand := "Db_Equipment".Compressor[7].IO.DO_Start,   // "FB_CompressorSim"
           OnFeedBack => "DB_Simulation".CompressorOnFb[7],
           OffFeedback => "DB_Simulation".CompressorOffFb[7]);
END_REGION

REGION Network 8
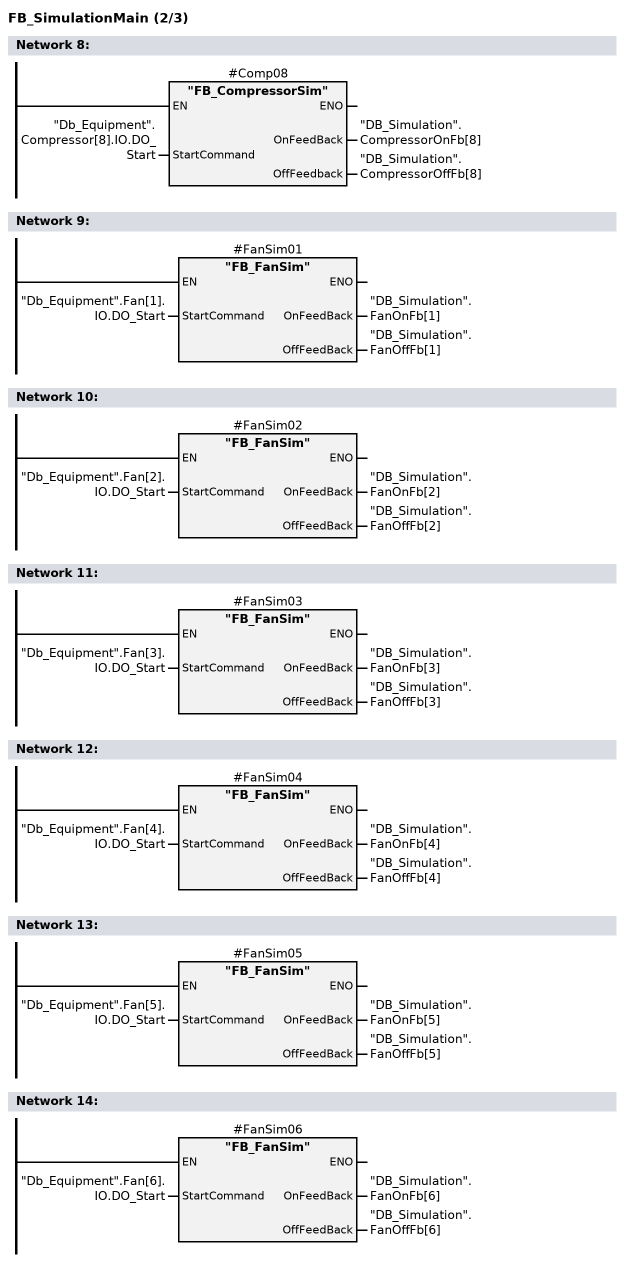
   RUNG wire#powerrail
      #Comp08(StartCommand := "Db_Equipment".Compressor[8].IO.DO_Start, OnFeedBack => "DB_Simulation".CompressorOnFb[8], OffFeedback => "DB_Simulation".CompressorOffFb[8])
   END_RUNG
   // the same network as SCL:
   #Comp08(StartCommand := "Db_Equipment".Compressor[8].IO.DO_Start,   // "FB_CompressorSim"
           OnFeedBack => "DB_Simulation".CompressorOnFb[8],
           OffFeedback => "DB_Simulation".CompressorOffFb[8]);
END_REGION

REGION Network 9
   RUNG wire#powerrail
      #FanSim01(StartCommand := "Db_Equipment".Fan[1].IO.DO_Start, OnFeedBack => "DB_Simulation".FanOnFb[1], OffFeedBack => "DB_Simulation".FanOffFb[1])
   END_RUNG
   // the same network as SCL:
   #FanSim01(StartCommand := "Db_Equipment".Fan[1].IO.DO_Start,   // "FB_FanSim"
             OnFeedBack => "DB_Simulation".FanOnFb[1],
             OffFeedBack => "DB_Simulation".FanOffFb[1]);
END_REGION

REGION Network 10
   RUNG wire#powerrail
      #FanSim02(StartCommand := "Db_Equipment".Fan[2].IO.DO_Start, OnFeedBack => "DB_Simulation".FanOnFb[2], OffFeedBack => "DB_Simulation".FanOffFb[2])
   END_RUNG
   // the same network as SCL:
   #FanSim02(StartCommand := "Db_Equipment".Fan[2].IO.DO_Start,   // "FB_FanSim"
             OnFeedBack => "DB_Simulation".FanOnFb[2],
             OffFeedBack => "DB_Simulation".FanOffFb[2]);
END_REGION

REGION Network 11
   RUNG wire#powerrail
      #FanSim03(StartCommand := "Db_Equipment".Fan[3].IO.DO_Start, OnFeedBack => "DB_Simulation".FanOnFb[3], OffFeedBack => "DB_Simulation".FanOffFb[3])
   END_RUNG
   // the same network as SCL:
   #FanSim03(StartCommand := "Db_Equipment".Fan[3].IO.DO_Start,   // "FB_FanSim"
             OnFeedBack => "DB_Simulation".FanOnFb[3],
             OffFeedBack => "DB_Simulation".FanOffFb[3]);
END_REGION

REGION Network 12
   RUNG wire#powerrail
      #FanSim04(StartCommand := "Db_Equipment".Fan[4].IO.DO_Start, OnFeedBack => "DB_Simulation".FanOnFb[4], OffFeedBack => "DB_Simulation".FanOffFb[4])
   END_RUNG
   // the same network as SCL:
   #FanSim04(StartCommand := "Db_Equipment".Fan[4].IO.DO_Start,   // "FB_FanSim"
             OnFeedBack => "DB_Simulation".FanOnFb[4],
             OffFeedBack => "DB_Simulation".FanOffFb[4]);
END_REGION

REGION Network 13
   RUNG wire#powerrail
      #FanSim05(StartCommand := "Db_Equipment".Fan[5].IO.DO_Start, OnFeedBack => "DB_Simulation".FanOnFb[5], OffFeedBack => "DB_Simulation".FanOffFb[5])
   END_RUNG
   // the same network as SCL:
   #FanSim05(StartCommand := "Db_Equipment".Fan[5].IO.DO_Start,   // "FB_FanSim"
             OnFeedBack => "DB_Simulation".FanOnFb[5],
             OffFeedBack => "DB_Simulation".FanOffFb[5]);
END_REGION

REGION Network 14
   RUNG wire#powerrail
      #FanSim06(StartCommand := "Db_Equipment".Fan[6].IO.DO_Start, OnFeedBack => "DB_Simulation".FanOnFb[6], OffFeedBack => "DB_Simulation".FanOffFb[6])
   END_RUNG
   // the same network as SCL:
   #FanSim06(StartCommand := "Db_Equipment".Fan[6].IO.DO_Start,   // "FB_FanSim"
             OnFeedBack => "DB_Simulation".FanOnFb[6],
             OffFeedBack => "DB_Simulation".FanOffFb[6]);
END_REGION

REGION Network 15
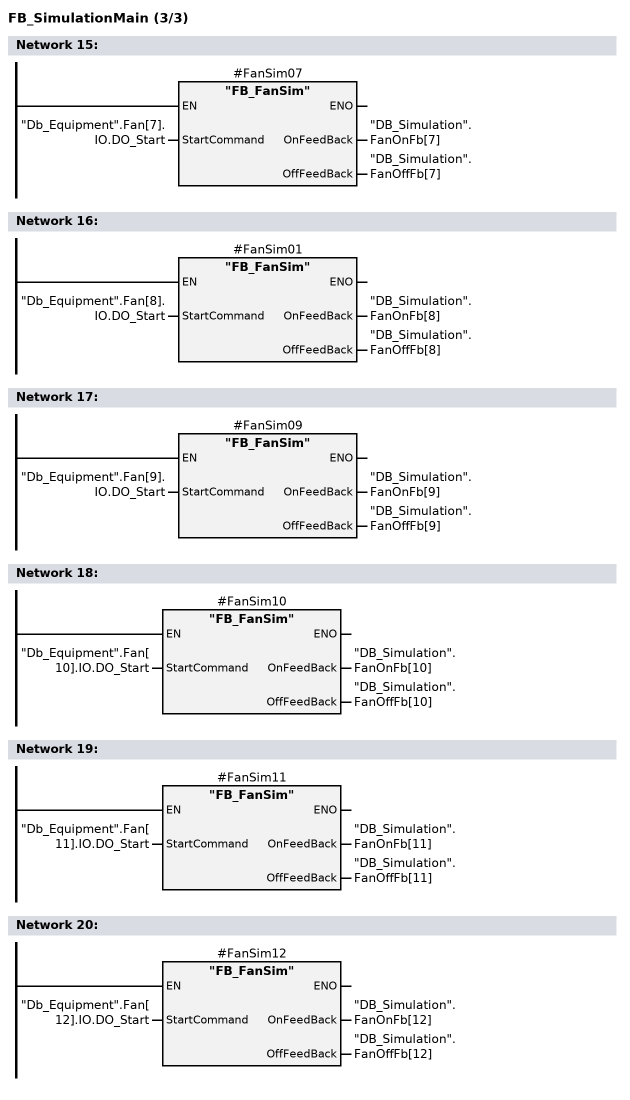
   RUNG wire#powerrail
      #FanSim07(StartCommand := "Db_Equipment".Fan[7].IO.DO_Start, OnFeedBack => "DB_Simulation".FanOnFb[7], OffFeedBack => "DB_Simulation".FanOffFb[7])
   END_RUNG
   // the same network as SCL:
   #FanSim07(StartCommand := "Db_Equipment".Fan[7].IO.DO_Start,   // "FB_FanSim"
             OnFeedBack => "DB_Simulation".FanOnFb[7],
             OffFeedBack => "DB_Simulation".FanOffFb[7]);
END_REGION

REGION Network 16
   RUNG wire#powerrail
      #FanSim01(StartCommand := "Db_Equipment".Fan[8].IO.DO_Start, OnFeedBack => "DB_Simulation".FanOnFb[8], OffFeedBack => "DB_Simulation".FanOffFb[8])
   END_RUNG
   // the same network as SCL:
   #FanSim01(StartCommand := "Db_Equipment".Fan[8].IO.DO_Start,   // "FB_FanSim"
             OnFeedBack => "DB_Simulation".FanOnFb[8],
             OffFeedBack => "DB_Simulation".FanOffFb[8]);
END_REGION

REGION Network 17
   RUNG wire#powerrail
      #FanSim09(StartCommand := "Db_Equipment".Fan[9].IO.DO_Start, OnFeedBack => "DB_Simulation".FanOnFb[9], OffFeedBack => "DB_Simulation".FanOffFb[9])
   END_RUNG
   // the same network as SCL:
   #FanSim09(StartCommand := "Db_Equipment".Fan[9].IO.DO_Start,   // "FB_FanSim"
             OnFeedBack => "DB_Simulation".FanOnFb[9],
             OffFeedBack => "DB_Simulation".FanOffFb[9]);
END_REGION

REGION Network 18
   RUNG wire#powerrail
      #FanSim10(StartCommand := "Db_Equipment".Fan[10].IO.DO_Start, OnFeedBack => "DB_Simulation".FanOnFb[10], OffFeedBack => "DB_Simulation".FanOffFb[10])
   END_RUNG
   // the same network as SCL:
   #FanSim10(StartCommand := "Db_Equipment".Fan[10].IO.DO_Start,   // "FB_FanSim"
             OnFeedBack => "DB_Simulation".FanOnFb[10],
             OffFeedBack => "DB_Simulation".FanOffFb[10]);
END_REGION

REGION Network 19
   RUNG wire#powerrail
      #FanSim11(StartCommand := "Db_Equipment".Fan[11].IO.DO_Start, OnFeedBack => "DB_Simulation".FanOnFb[11], OffFeedBack => "DB_Simulation".FanOffFb[11])
   END_RUNG
   // the same network as SCL:
   #FanSim11(StartCommand := "Db_Equipment".Fan[11].IO.DO_Start,   // "FB_FanSim"
             OnFeedBack => "DB_Simulation".FanOnFb[11],
             OffFeedBack => "DB_Simulation".FanOffFb[11]);
END_REGION

REGION Network 20
   RUNG wire#powerrail
      #FanSim12(StartCommand := "Db_Equipment".Fan[12].IO.DO_Start, OnFeedBack => "DB_Simulation".FanOnFb[12], OffFeedBack => "DB_Simulation".FanOffFb[12])
   END_RUNG
   // the same network as SCL:
   #FanSim12(StartCommand := "Db_Equipment".Fan[12].IO.DO_Start,   // "FB_FanSim"
             OnFeedBack => "DB_Simulation".FanOnFb[12],
             OffFeedBack => "DB_Simulation".FanOffFb[12]);
END_REGION
END_FUNCTION_BLOCK

ORGANIZATION_BLOCK "OB1_Main"   // OB1, LAD, ProgramCycle
TITLE = "Main Program Sweep (Cycle)"
{ S7_Optimized_Access := 'TRUE' }
VERSION : 0.1
   VAR_INPUT
      Initial_Call : Bool;   // Initial call of this OB
      Remanence : Bool;   // =True, if remanent data are available
   END_VAR
BEGIN

REGION Network 1
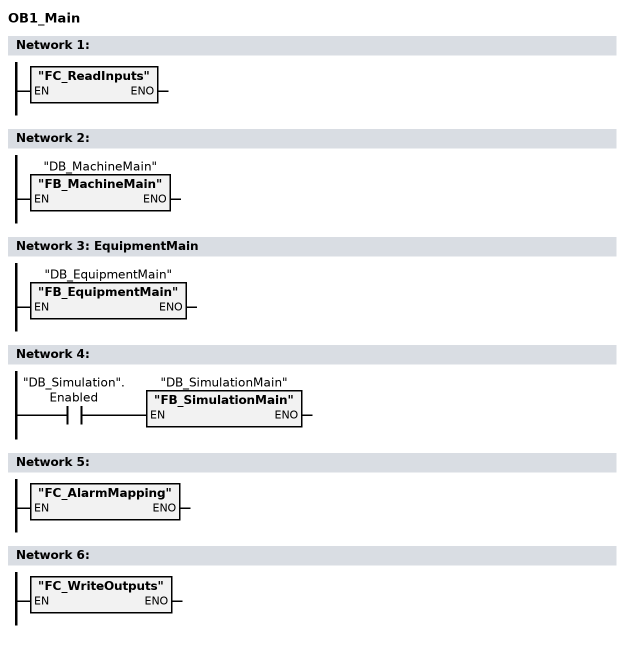
   RUNG wire#powerrail
      "FC_ReadInputs"()
   END_RUNG
   // the same network as SCL:
   "FC_ReadInputs"();
END_REGION

REGION Network 2
   RUNG wire#powerrail
      "DB_MachineMain"()
   END_RUNG
   // the same network as SCL:
   "DB_MachineMain"();   // "FB_MachineMain"
END_REGION

REGION Network 3: EquipmentMain
   RUNG wire#powerrail
      "DB_EquipmentMain"()
   END_RUNG
   // the same network as SCL:
   "DB_EquipmentMain"();   // "FB_EquipmentMain"
END_REGION

REGION Network 4
   RUNG wire#powerrail
      Contact( "DB_Simulation".Enabled )
      "DB_SimulationMain"()
   END_RUNG
   // the same network as SCL:
   IF "DB_Simulation".Enabled THEN
       "DB_SimulationMain"();   // "FB_SimulationMain"
   END_IF;
END_REGION

REGION Network 5
   RUNG wire#powerrail
      "FC_AlarmMapping"()
   END_RUNG
   // the same network as SCL:
   "FC_AlarmMapping"();
END_REGION

REGION Network 6
   RUNG wire#powerrail
      "FC_WriteOutputs"()
   END_RUNG
   // the same network as SCL:
   "FC_WriteOutputs"();
END_REGION
END_ORGANIZATION_BLOCK

ORGANIZATION_BLOCK "0B30_PID"   // OB30, LAD, CyclicInterrupt
{ S7_Optimized_Access := 'TRUE' }
VERSION : 0.1
   VAR_INPUT
      Initial_Call : Bool;   // Initial call of this OB
      Event_Count : Int;   // Events discarded
   END_VAR
BEGIN

REGION Network 1
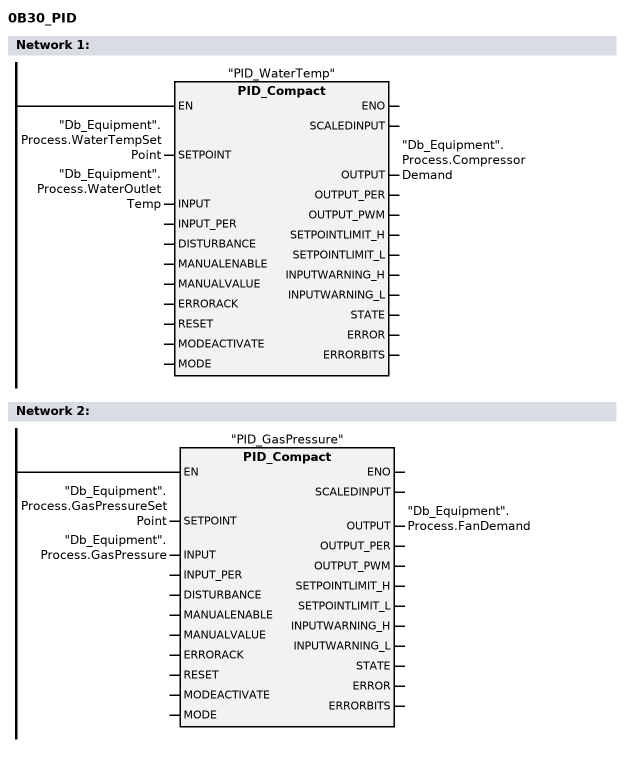
   "PID_WaterTemp"(Setpoint := "Db_Equipment".Process.WaterTempSetPoint,   // PID_Compact
                   Input := "Db_Equipment".Process.WaterOutletTemp,
                   Output => "Db_Equipment".Process.CompressorDemand);
END_REGION

REGION Network 2
   "PID_GasPressure"(Setpoint := "Db_Equipment".Process.GasPressureSetPoint,   // PID_Compact
                     Input := "Db_Equipment".Process.GasPressure,
                     Output => "Db_Equipment".Process.FanDemand);
END_REGION
END_ORGANIZATION_BLOCK

// folder: 01_equitmen

FUNCTION_BLOCK "FB_Compressor"   // FB1, LAD
{ S7_Optimized_Access := 'TRUE' }
VERSION : 0.1
   VAR_INPUT
      Timing : "UDT_TimingParams";
   END_VAR
   VAR_IN_OUT
      Comp : "UDT_Compressor";
   END_VAR
   VAR
      StartLatch : Bool;
      tFeedback : TON_TIME;
      tMinOn : TON_TIME;
      tMinOff : TON_TIME;
      RuntimeEdge : Bool;
   END_VAR
   VAR_TEMP
      MinOffDone : Bool;
      MinOnDone : Bool;
      StopCondition : Bool;
      FeedbackTimeout : Bool;
      RunSecondsReal : Real;
   END_VAR
   VAR_TEMP   // added for the SCL form of the ladder/FBD networks
      _w1 : Bool;
   END_VAR
BEGIN

REGION Network 1: Fault Calculation
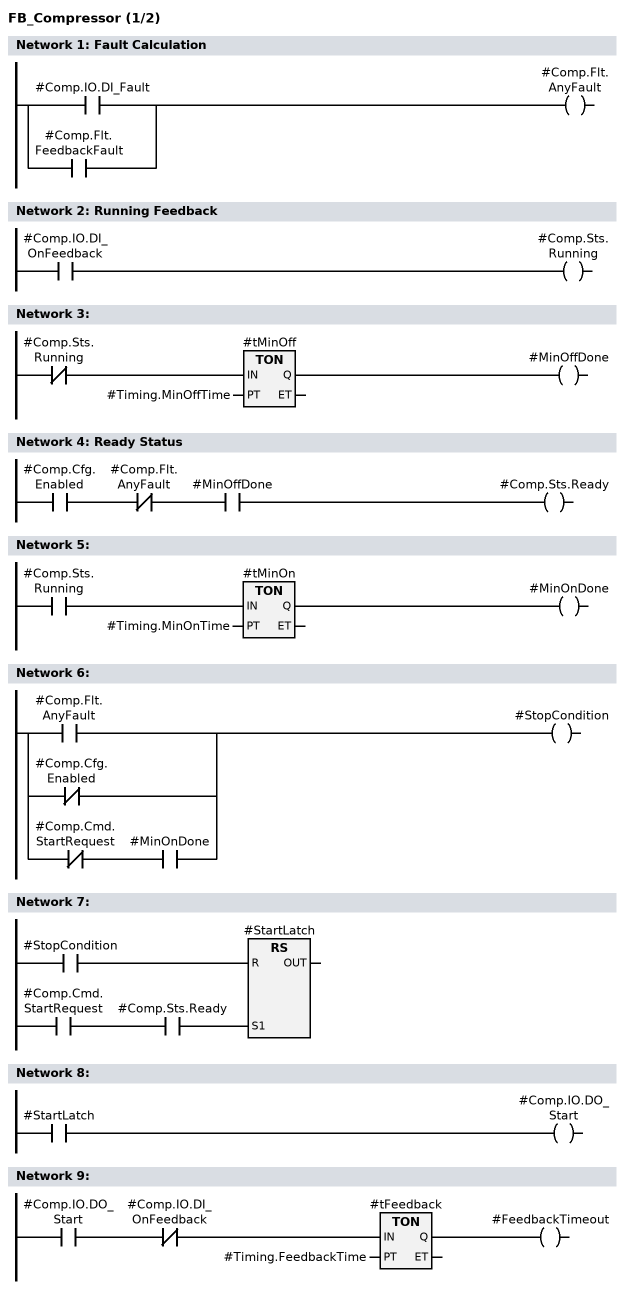
   RUNG wire#powerrail
      Contact( #Comp.IO.DI_Fault )
      wire#w1
      Coil( #Comp.Flt.AnyFault )
   END_RUNG
   RUNG wire#powerrail
      Contact( #Comp.Flt.FeedbackFault )
   END_RUNG wire#w1
   // the same network as SCL:
   #Comp.Flt.AnyFault := #Comp.IO.DI_Fault OR #Comp.Flt.FeedbackFault;
END_REGION

REGION Network 2: Running Feedback
   RUNG wire#powerrail
      Contact( #Comp.IO.DI_OnFeedback )
      Coil( #Comp.Sts.Running )
   END_RUNG
   // the same network as SCL:
   #Comp.Sts.Running := #Comp.IO.DI_OnFeedback;
END_REGION

REGION Network 3
   #tMinOff(IN := NOT #Comp.Sts.Running, PT := #Timing.MinOffTime);   // TON
   #MinOffDone := #tMinOff.Q;
END_REGION

REGION Network 4: Ready Status
   RUNG wire#powerrail
      Contact( #Comp.Cfg.Enabled )
      I_Contact( #Comp.Flt.AnyFault )
      Contact( #MinOffDone )
      Coil( #Comp.Sts.Ready )
   END_RUNG
   // the same network as SCL:
   #Comp.Sts.Ready := #Comp.Cfg.Enabled AND NOT #Comp.Flt.AnyFault AND #MinOffDone;
END_REGION

REGION Network 5
   #tMinOn(IN := #Comp.Sts.Running, PT := #Timing.MinOnTime);   // TON
   #MinOnDone := #tMinOn.Q;
END_REGION

REGION Network 6
   RUNG wire#powerrail
      Contact( #Comp.Flt.AnyFault )
      wire#w1
      Coil( #StopCondition )
   END_RUNG
   RUNG wire#powerrail
      I_Contact( #Comp.Cfg.Enabled )
   END_RUNG wire#w1
   RUNG wire#powerrail
      I_Contact( #Comp.Cmd.StartRequest )
      Contact( #MinOnDone )
   END_RUNG wire#w1
   // the same network as SCL:
   #StopCondition := #Comp.Flt.AnyFault OR NOT #Comp.Cfg.Enabled OR (NOT #Comp.Cmd.StartRequest AND #MinOnDone);
END_REGION

REGION Network 7
   RUNG wire#powerrail
      Contact( #StopCondition )
      S_RS(operand := #StartLatch, s1 := wire#w1)
   END_RUNG
   RUNG wire#powerrail
      Contact( #Comp.Cmd.StartRequest )
      Contact( #Comp.Sts.Ready )
   END_RUNG wire#w1
   // the same network as SCL:
   IF #StopCondition THEN
       #StartLatch := FALSE;   // RS flip-flop
   END_IF;
   IF #Comp.Cmd.StartRequest AND #Comp.Sts.Ready THEN #StartLatch := TRUE; END_IF;
END_REGION

REGION Network 8
   RUNG wire#powerrail
      Contact( #StartLatch )
      Coil( #Comp.IO.DO_Start )
   END_RUNG
   // the same network as SCL:
   #Comp.IO.DO_Start := #StartLatch;
END_REGION

REGION Network 9
   #tFeedback(IN := #Comp.IO.DO_Start AND NOT #Comp.IO.DI_OnFeedback, PT := #Timing.FeedbackTime);   // TON
   #FeedbackTimeout := #tFeedback.Q;
END_REGION

REGION Network 10
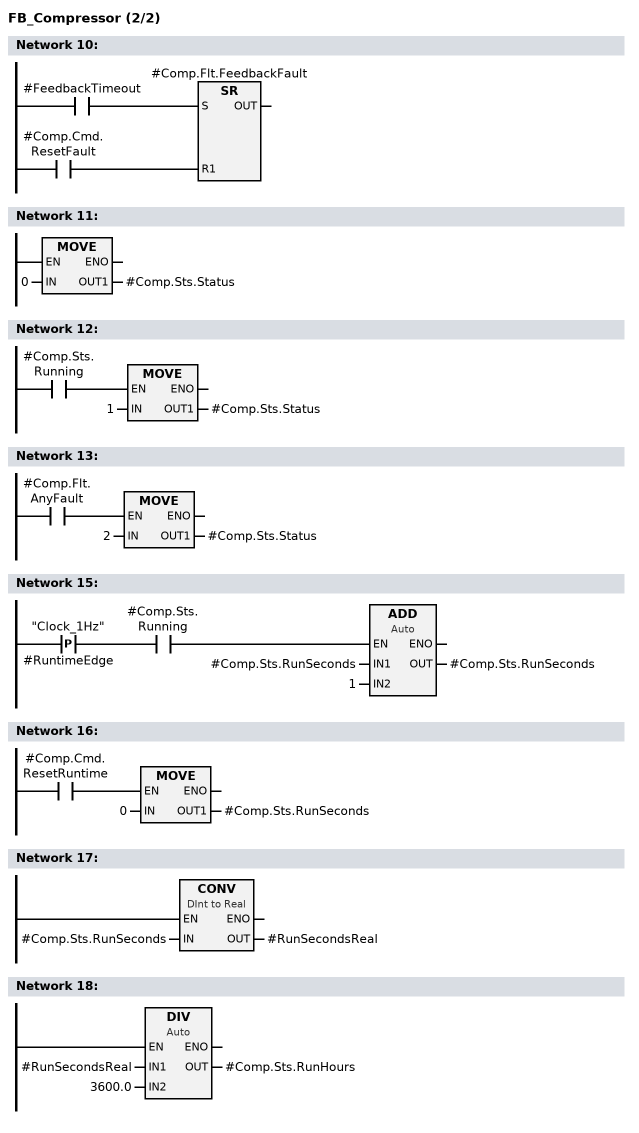
   RUNG wire#powerrail
      Contact( #FeedbackTimeout )
      S_SR(operand := #Comp.Flt.FeedbackFault, r1 := wire#w1)
   END_RUNG
   RUNG wire#powerrail
      Contact( #Comp.Cmd.ResetFault )
   END_RUNG wire#w1
   // the same network as SCL:
   IF #FeedbackTimeout THEN
       #Comp.Flt.FeedbackFault := TRUE;   // SR flip-flop
   END_IF;
   IF #Comp.Cmd.ResetFault THEN #Comp.Flt.FeedbackFault := FALSE; END_IF;
END_REGION

REGION Network 11
   RUNG wire#powerrail
      Move(in := 0, out1 => #Comp.Sts.Status)
   END_RUNG
   // the same network as SCL:
   #Comp.Sts.Status := 0;
END_REGION

REGION Network 12
   RUNG wire#powerrail
      Contact( #Comp.Sts.Running )
      Move(in := 1, out1 => #Comp.Sts.Status)
   END_RUNG
   // the same network as SCL:
   IF #Comp.Sts.Running THEN #Comp.Sts.Status := 1; END_IF;
END_REGION

REGION Network 13
   RUNG wire#powerrail
      Contact( #Comp.Flt.AnyFault )
      Move(in := 2, out1 => #Comp.Sts.Status)
   END_RUNG
   // the same network as SCL:
   IF #Comp.Flt.AnyFault THEN #Comp.Sts.Status := 2; END_IF;
END_REGION

REGION Network 15
   RUNG wire#powerrail
      P_Contact(operand := "Clock_1Hz", bit := #RuntimeEdge)
      Contact( #Comp.Sts.Running )
      Add(in1 := #Comp.Sts.RunSeconds, in2 := 1, out => #Comp.Sts.RunSeconds)
   END_RUNG
   // the same network as SCL:
   #_w1 := "Clock_1Hz" AND NOT #RuntimeEdge;   // rising edge of "Clock_1Hz"
   #RuntimeEdge := "Clock_1Hz";
   IF #_w1 AND #Comp.Sts.Running THEN #Comp.Sts.RunSeconds := #Comp.Sts.RunSeconds + 1; END_IF;
END_REGION

REGION Network 16
   RUNG wire#powerrail
      Contact( #Comp.Cmd.ResetRuntime )
      Move(in := 0, out1 => #Comp.Sts.RunSeconds)
   END_RUNG
   // the same network as SCL:
   IF #Comp.Cmd.ResetRuntime THEN #Comp.Sts.RunSeconds := 0; END_IF;
END_REGION

REGION Network 17
   RUNG wire#powerrail
      { S7_Templates := "[SrcType := DInt, DestType := Real]" } Convert(in := #Comp.Sts.RunSeconds, out => #RunSecondsReal)
   END_RUNG
   // the same network as SCL:
   #RunSecondsReal := DINT_TO_REAL(#Comp.Sts.RunSeconds);
END_REGION

REGION Network 18
   RUNG wire#powerrail
      Div(in1 := #RunSecondsReal, in2 := 3600.0, out => #Comp.Sts.RunHours)
   END_RUNG
   // the same network as SCL:
   #Comp.Sts.RunHours := #RunSecondsReal / 3600.0;
END_REGION
END_FUNCTION_BLOCK

FUNCTION_BLOCK "FB_CompressorManager"   // FB2, LAD
{ S7_Optimized_Access := 'TRUE' }
VERSION : 0.1
   VAR_INPUT
      RequiredCount : Int;
   END_VAR
   VAR_OUTPUT
      RunningCount : Int;
      RequestCount : Int;
   END_VAR
   VAR_IN_OUT
      Comp : Array[1..8] of "UDT_Compressor";
   END_VAR
   VAR_TEMP
      StartCandidate : Int;
      StopCandidate : Int;
      MinRuntime : DInt;
      MaxRunTime : DInt;
      StartRequired : Bool;
      StopRequired : Bool;
   END_VAR
   VAR_TEMP   // added for the SCL form of the ladder/FBD networks
      _w1 : Bool;
   END_VAR
BEGIN

REGION Network 1
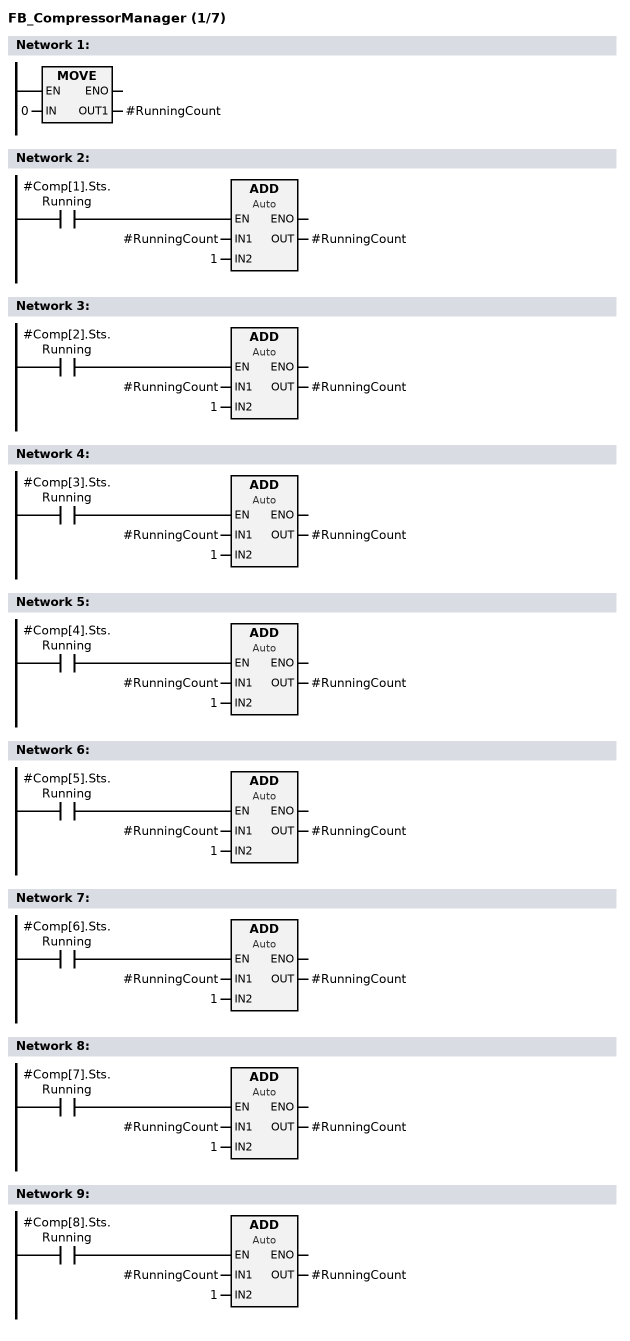
   RUNG wire#powerrail
      Move(in := 0, out1 => #RunningCount)
   END_RUNG
   // the same network as SCL:
   #RunningCount := 0;
END_REGION

REGION Network 2
   RUNG wire#powerrail
      Contact( #Comp[1].Sts.Running )
      Add(in1 := #RunningCount, in2 := 1, out => #RunningCount)
   END_RUNG
   // the same network as SCL:
   IF #Comp[1].Sts.Running THEN #RunningCount := #RunningCount + 1; END_IF;
END_REGION

REGION Network 3
   RUNG wire#powerrail
      Contact( #Comp[2].Sts.Running )
      Add(in1 := #RunningCount, in2 := 1, out => #RunningCount)
   END_RUNG
   // the same network as SCL:
   IF #Comp[2].Sts.Running THEN #RunningCount := #RunningCount + 1; END_IF;
END_REGION

REGION Network 4
   RUNG wire#powerrail
      Contact( #Comp[3].Sts.Running )
      Add(in1 := #RunningCount, in2 := 1, out => #RunningCount)
   END_RUNG
   // the same network as SCL:
   IF #Comp[3].Sts.Running THEN #RunningCount := #RunningCount + 1; END_IF;
END_REGION

REGION Network 5
   RUNG wire#powerrail
      Contact( #Comp[4].Sts.Running )
      Add(in1 := #RunningCount, in2 := 1, out => #RunningCount)
   END_RUNG
   // the same network as SCL:
   IF #Comp[4].Sts.Running THEN #RunningCount := #RunningCount + 1; END_IF;
END_REGION

REGION Network 6
   RUNG wire#powerrail
      Contact( #Comp[5].Sts.Running )
      Add(in1 := #RunningCount, in2 := 1, out => #RunningCount)
   END_RUNG
   // the same network as SCL:
   IF #Comp[5].Sts.Running THEN #RunningCount := #RunningCount + 1; END_IF;
END_REGION

REGION Network 7
   RUNG wire#powerrail
      Contact( #Comp[6].Sts.Running )
      Add(in1 := #RunningCount, in2 := 1, out => #RunningCount)
   END_RUNG
   // the same network as SCL:
   IF #Comp[6].Sts.Running THEN #RunningCount := #RunningCount + 1; END_IF;
END_REGION

REGION Network 8
   RUNG wire#powerrail
      Contact( #Comp[7].Sts.Running )
      Add(in1 := #RunningCount, in2 := 1, out => #RunningCount)
   END_RUNG
   // the same network as SCL:
   IF #Comp[7].Sts.Running THEN #RunningCount := #RunningCount + 1; END_IF;
END_REGION

REGION Network 9
   RUNG wire#powerrail
      Contact( #Comp[8].Sts.Running )
      Add(in1 := #RunningCount, in2 := 1, out => #RunningCount)
   END_RUNG
   // the same network as SCL:
   IF #Comp[8].Sts.Running THEN #RunningCount := #RunningCount + 1; END_IF;
END_REGION

REGION Network 10
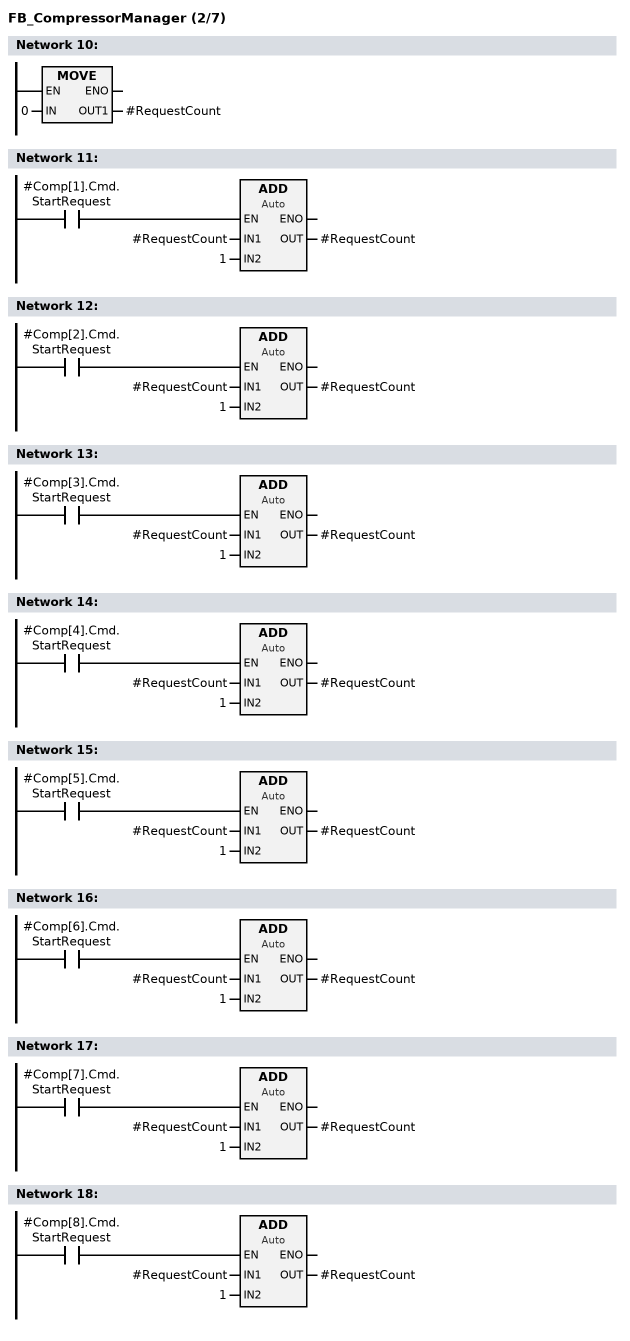
   RUNG wire#powerrail
      Move(in := 0, out1 => #RequestCount)
   END_RUNG
   // the same network as SCL:
   #RequestCount := 0;
END_REGION

REGION Network 11
   RUNG wire#powerrail
      Contact( #Comp[1].Cmd.StartRequest )
      Add(in1 := #RequestCount, in2 := 1, out => #RequestCount)
   END_RUNG
   // the same network as SCL:
   IF #Comp[1].Cmd.StartRequest THEN #RequestCount := #RequestCount + 1; END_IF;
END_REGION

REGION Network 12
   RUNG wire#powerrail
      Contact( #Comp[2].Cmd.StartRequest )
      Add(in1 := #RequestCount, in2 := 1, out => #RequestCount)
   END_RUNG
   // the same network as SCL:
   IF #Comp[2].Cmd.StartRequest THEN #RequestCount := #RequestCount + 1; END_IF;
END_REGION

REGION Network 13
   RUNG wire#powerrail
      Contact( #Comp[3].Cmd.StartRequest )
      Add(in1 := #RequestCount, in2 := 1, out => #RequestCount)
   END_RUNG
   // the same network as SCL:
   IF #Comp[3].Cmd.StartRequest THEN #RequestCount := #RequestCount + 1; END_IF;
END_REGION

REGION Network 14
   RUNG wire#powerrail
      Contact( #Comp[4].Cmd.StartRequest )
      Add(in1 := #RequestCount, in2 := 1, out => #RequestCount)
   END_RUNG
   // the same network as SCL:
   IF #Comp[4].Cmd.StartRequest THEN #RequestCount := #RequestCount + 1; END_IF;
END_REGION

REGION Network 15
   RUNG wire#powerrail
      Contact( #Comp[5].Cmd.StartRequest )
      Add(in1 := #RequestCount, in2 := 1, out => #RequestCount)
   END_RUNG
   // the same network as SCL:
   IF #Comp[5].Cmd.StartRequest THEN #RequestCount := #RequestCount + 1; END_IF;
END_REGION

REGION Network 16
   RUNG wire#powerrail
      Contact( #Comp[6].Cmd.StartRequest )
      Add(in1 := #RequestCount, in2 := 1, out => #RequestCount)
   END_RUNG
   // the same network as SCL:
   IF #Comp[6].Cmd.StartRequest THEN #RequestCount := #RequestCount + 1; END_IF;
END_REGION

REGION Network 17
   RUNG wire#powerrail
      Contact( #Comp[7].Cmd.StartRequest )
      Add(in1 := #RequestCount, in2 := 1, out => #RequestCount)
   END_RUNG
   // the same network as SCL:
   IF #Comp[7].Cmd.StartRequest THEN #RequestCount := #RequestCount + 1; END_IF;
END_REGION

REGION Network 18
   RUNG wire#powerrail
      Contact( #Comp[8].Cmd.StartRequest )
      Add(in1 := #RequestCount, in2 := 1, out => #RequestCount)
   END_RUNG
   // the same network as SCL:
   IF #Comp[8].Cmd.StartRequest THEN #RequestCount := #RequestCount + 1; END_IF;
END_REGION

REGION Network 19
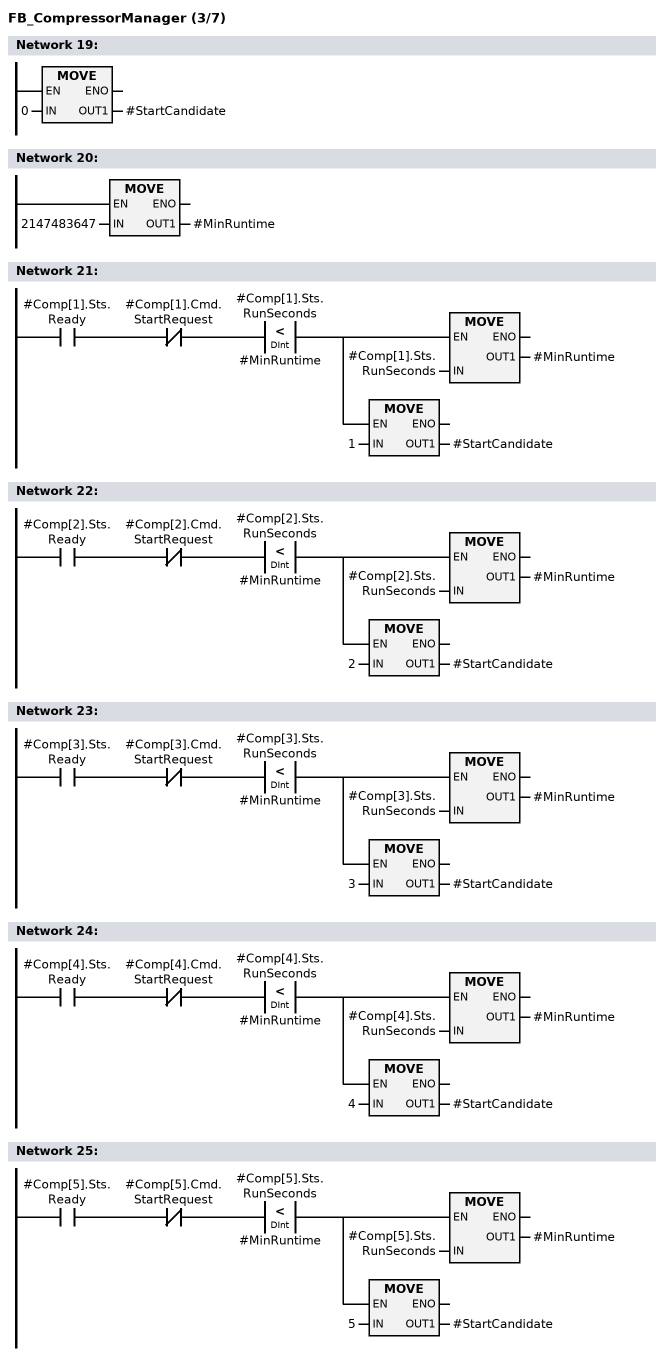
   RUNG wire#powerrail
      Move(in := 0, out1 => #StartCandidate)
   END_RUNG
   // the same network as SCL:
   #StartCandidate := 0;
END_REGION

REGION Network 20
   RUNG wire#powerrail
      Move(in := 2147483647, out1 => #MinRuntime)
   END_RUNG
   // the same network as SCL:
   #MinRuntime := 2147483647;
END_REGION

REGION Network 21
   RUNG wire#powerrail
      Contact( #Comp[1].Sts.Ready )
      I_Contact( #Comp[1].Cmd.StartRequest )
      { S7_Templates := "SrcType := DInt" } LT_Contact(in1 := #Comp[1].Sts.RunSeconds, in2 := #MinRuntime)
      wire#w1
      Move(in := #Comp[1].Sts.RunSeconds, out1 => #MinRuntime)
   END_RUNG
   RUNG wire#w1
      Move(in := 1, out1 => #StartCandidate)
   END_RUNG
   // the same network as SCL:
   #_w1 := #Comp[1].Sts.Ready AND NOT #Comp[1].Cmd.StartRequest AND (#Comp[1].Sts.RunSeconds < #MinRuntime);
   IF #_w1 THEN
       #MinRuntime := #Comp[1].Sts.RunSeconds;
       #StartCandidate := 1;
   END_IF;
END_REGION

REGION Network 22
   RUNG wire#powerrail
      Contact( #Comp[2].Sts.Ready )
      I_Contact( #Comp[2].Cmd.StartRequest )
      { S7_Templates := "SrcType := DInt" } LT_Contact(in1 := #Comp[2].Sts.RunSeconds, in2 := #MinRuntime)
      wire#w1
      Move(in := #Comp[2].Sts.RunSeconds, out1 => #MinRuntime)
   END_RUNG
   RUNG wire#w1
      Move(in := 2, out1 => #StartCandidate)
   END_RUNG
   // the same network as SCL:
   #_w1 := #Comp[2].Sts.Ready AND NOT #Comp[2].Cmd.StartRequest AND (#Comp[2].Sts.RunSeconds < #MinRuntime);
   IF #_w1 THEN
       #MinRuntime := #Comp[2].Sts.RunSeconds;
       #StartCandidate := 2;
   END_IF;
END_REGION

REGION Network 23
   RUNG wire#powerrail
      Contact( #Comp[3].Sts.Ready )
      I_Contact( #Comp[3].Cmd.StartRequest )
      { S7_Templates := "SrcType := DInt" } LT_Contact(in1 := #Comp[3].Sts.RunSeconds, in2 := #MinRuntime)
      wire#w1
      Move(in := #Comp[3].Sts.RunSeconds, out1 => #MinRuntime)
   END_RUNG
   RUNG wire#w1
      Move(in := 3, out1 => #StartCandidate)
   END_RUNG
   // the same network as SCL:
   #_w1 := #Comp[3].Sts.Ready AND NOT #Comp[3].Cmd.StartRequest AND (#Comp[3].Sts.RunSeconds < #MinRuntime);
   IF #_w1 THEN
       #MinRuntime := #Comp[3].Sts.RunSeconds;
       #StartCandidate := 3;
   END_IF;
END_REGION

REGION Network 24
   RUNG wire#powerrail
      Contact( #Comp[4].Sts.Ready )
      I_Contact( #Comp[4].Cmd.StartRequest )
      { S7_Templates := "SrcType := DInt" } LT_Contact(in1 := #Comp[4].Sts.RunSeconds, in2 := #MinRuntime)
      wire#w1
      Move(in := #Comp[4].Sts.RunSeconds, out1 => #MinRuntime)
   END_RUNG
   RUNG wire#w1
      Move(in := 4, out1 => #StartCandidate)
   END_RUNG
   // the same network as SCL:
   #_w1 := #Comp[4].Sts.Ready AND NOT #Comp[4].Cmd.StartRequest AND (#Comp[4].Sts.RunSeconds < #MinRuntime);
   IF #_w1 THEN
       #MinRuntime := #Comp[4].Sts.RunSeconds;
       #StartCandidate := 4;
   END_IF;
END_REGION

REGION Network 25
   RUNG wire#powerrail
      Contact( #Comp[5].Sts.Ready )
      I_Contact( #Comp[5].Cmd.StartRequest )
      { S7_Templates := "SrcType := DInt" } LT_Contact(in1 := #Comp[5].Sts.RunSeconds, in2 := #MinRuntime)
      wire#w1
      Move(in := #Comp[5].Sts.RunSeconds, out1 => #MinRuntime)
   END_RUNG
   RUNG wire#w1
      Move(in := 5, out1 => #StartCandidate)
   END_RUNG
   // the same network as SCL:
   #_w1 := #Comp[5].Sts.Ready AND NOT #Comp[5].Cmd.StartRequest AND (#Comp[5].Sts.RunSeconds < #MinRuntime);
   IF #_w1 THEN
       #MinRuntime := #Comp[5].Sts.RunSeconds;
       #StartCandidate := 5;
   END_IF;
END_REGION

REGION Network 26
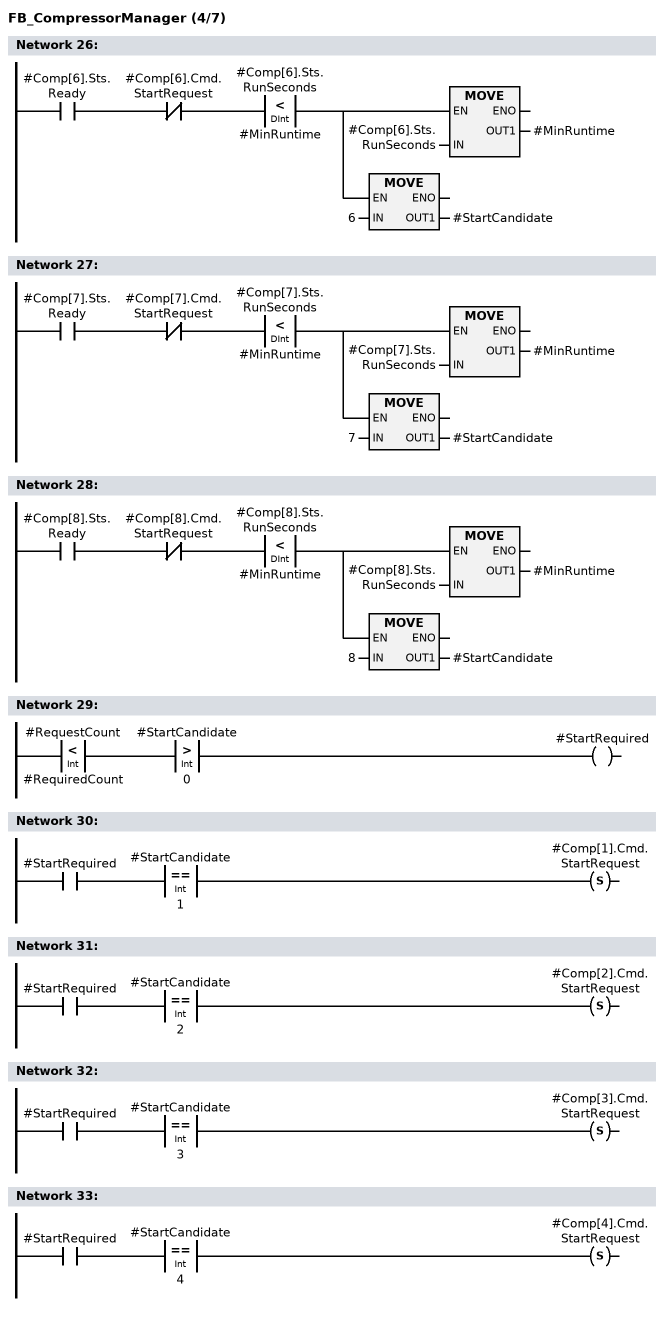
   RUNG wire#powerrail
      Contact( #Comp[6].Sts.Ready )
      I_Contact( #Comp[6].Cmd.StartRequest )
      { S7_Templates := "SrcType := DInt" } LT_Contact(in1 := #Comp[6].Sts.RunSeconds, in2 := #MinRuntime)
      wire#w1
      Move(in := #Comp[6].Sts.RunSeconds, out1 => #MinRuntime)
   END_RUNG
   RUNG wire#w1
      Move(in := 6, out1 => #StartCandidate)
   END_RUNG
   // the same network as SCL:
   #_w1 := #Comp[6].Sts.Ready AND NOT #Comp[6].Cmd.StartRequest AND (#Comp[6].Sts.RunSeconds < #MinRuntime);
   IF #_w1 THEN
       #MinRuntime := #Comp[6].Sts.RunSeconds;
       #StartCandidate := 6;
   END_IF;
END_REGION

REGION Network 27
   RUNG wire#powerrail
      Contact( #Comp[7].Sts.Ready )
      I_Contact( #Comp[7].Cmd.StartRequest )
      { S7_Templates := "SrcType := DInt" } LT_Contact(in1 := #Comp[7].Sts.RunSeconds, in2 := #MinRuntime)
      wire#w1
      Move(in := #Comp[7].Sts.RunSeconds, out1 => #MinRuntime)
   END_RUNG
   RUNG wire#w1
      Move(in := 7, out1 => #StartCandidate)
   END_RUNG
   // the same network as SCL:
   #_w1 := #Comp[7].Sts.Ready AND NOT #Comp[7].Cmd.StartRequest AND (#Comp[7].Sts.RunSeconds < #MinRuntime);
   IF #_w1 THEN
       #MinRuntime := #Comp[7].Sts.RunSeconds;
       #StartCandidate := 7;
   END_IF;
END_REGION

REGION Network 28
   RUNG wire#powerrail
      Contact( #Comp[8].Sts.Ready )
      I_Contact( #Comp[8].Cmd.StartRequest )
      { S7_Templates := "SrcType := DInt" } LT_Contact(in1 := #Comp[8].Sts.RunSeconds, in2 := #MinRuntime)
      wire#w1
      Move(in := #Comp[8].Sts.RunSeconds, out1 => #MinRuntime)
   END_RUNG
   RUNG wire#w1
      Move(in := 8, out1 => #StartCandidate)
   END_RUNG
   // the same network as SCL:
   #_w1 := #Comp[8].Sts.Ready AND NOT #Comp[8].Cmd.StartRequest AND (#Comp[8].Sts.RunSeconds < #MinRuntime);
   IF #_w1 THEN
       #MinRuntime := #Comp[8].Sts.RunSeconds;
       #StartCandidate := 8;
   END_IF;
END_REGION

REGION Network 29
   RUNG wire#powerrail
      { S7_Templates := "SrcType := Int" } LT_Contact(in1 := #RequestCount, in2 := #RequiredCount)
      { S7_Templates := "SrcType := Int" } GT_Contact(in1 := #StartCandidate, in2 := 0)
      Coil( #StartRequired )
   END_RUNG
   // the same network as SCL:
   #StartRequired := (#RequestCount < #RequiredCount) AND (#StartCandidate > 0);
END_REGION

REGION Network 30
   RUNG wire#powerrail
      Contact( #StartRequired )
      { S7_Templates := "SrcType := Int" } EQ_Contact(in1 := #StartCandidate, in2 := 1)
      S_Coil( #Comp[1].Cmd.StartRequest )
   END_RUNG
   // the same network as SCL:
   IF #StartRequired AND (#StartCandidate = 1) THEN #Comp[1].Cmd.StartRequest := TRUE; END_IF;
END_REGION

REGION Network 31
   RUNG wire#powerrail
      Contact( #StartRequired )
      { S7_Templates := "SrcType := Int" } EQ_Contact(in1 := #StartCandidate, in2 := 2)
      S_Coil( #Comp[2].Cmd.StartRequest )
   END_RUNG
   // the same network as SCL:
   IF #StartRequired AND (#StartCandidate = 2) THEN #Comp[2].Cmd.StartRequest := TRUE; END_IF;
END_REGION

REGION Network 32
   RUNG wire#powerrail
      Contact( #StartRequired )
      { S7_Templates := "SrcType := Int" } EQ_Contact(in1 := #StartCandidate, in2 := 3)
      S_Coil( #Comp[3].Cmd.StartRequest )
   END_RUNG
   // the same network as SCL:
   IF #StartRequired AND (#StartCandidate = 3) THEN #Comp[3].Cmd.StartRequest := TRUE; END_IF;
END_REGION

REGION Network 33
   RUNG wire#powerrail
      Contact( #StartRequired )
      { S7_Templates := "SrcType := Int" } EQ_Contact(in1 := #StartCandidate, in2 := 4)
      S_Coil( #Comp[4].Cmd.StartRequest )
   END_RUNG
   // the same network as SCL:
   IF #StartRequired AND (#StartCandidate = 4) THEN #Comp[4].Cmd.StartRequest := TRUE; END_IF;
END_REGION

REGION Network 34
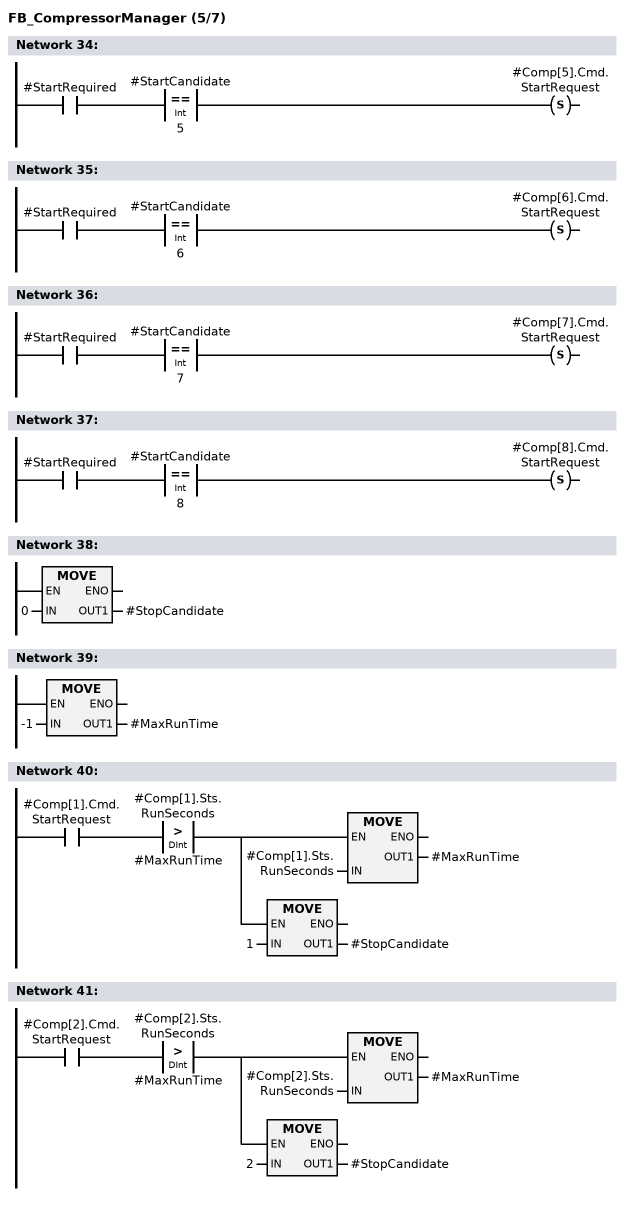
   RUNG wire#powerrail
      Contact( #StartRequired )
      { S7_Templates := "SrcType := Int" } EQ_Contact(in1 := #StartCandidate, in2 := 5)
      S_Coil( #Comp[5].Cmd.StartRequest )
   END_RUNG
   // the same network as SCL:
   IF #StartRequired AND (#StartCandidate = 5) THEN #Comp[5].Cmd.StartRequest := TRUE; END_IF;
END_REGION

REGION Network 35
   RUNG wire#powerrail
      Contact( #StartRequired )
      { S7_Templates := "SrcType := Int" } EQ_Contact(in1 := #StartCandidate, in2 := 6)
      S_Coil( #Comp[6].Cmd.StartRequest )
   END_RUNG
   // the same network as SCL:
   IF #StartRequired AND (#StartCandidate = 6) THEN #Comp[6].Cmd.StartRequest := TRUE; END_IF;
END_REGION

REGION Network 36
   RUNG wire#powerrail
      Contact( #StartRequired )
      { S7_Templates := "SrcType := Int" } EQ_Contact(in1 := #StartCandidate, in2 := 7)
      S_Coil( #Comp[7].Cmd.StartRequest )
   END_RUNG
   // the same network as SCL:
   IF #StartRequired AND (#StartCandidate = 7) THEN #Comp[7].Cmd.StartRequest := TRUE; END_IF;
END_REGION

REGION Network 37
   RUNG wire#powerrail
      Contact( #StartRequired )
      { S7_Templates := "SrcType := Int" } EQ_Contact(in1 := #StartCandidate, in2 := 8)
      S_Coil( #Comp[8].Cmd.StartRequest )
   END_RUNG
   // the same network as SCL:
   IF #StartRequired AND (#StartCandidate = 8) THEN #Comp[8].Cmd.StartRequest := TRUE; END_IF;
END_REGION

REGION Network 38
   RUNG wire#powerrail
      Move(in := 0, out1 => #StopCandidate)
   END_RUNG
   // the same network as SCL:
   #StopCandidate := 0;
END_REGION

REGION Network 39
   RUNG wire#powerrail
      Move(in := -1, out1 => #MaxRunTime)
   END_RUNG
   // the same network as SCL:
   #MaxRunTime := -1;
END_REGION

REGION Network 40
   RUNG wire#powerrail
      Contact( #Comp[1].Cmd.StartRequest )
      { S7_Templates := "SrcType := DInt" } GT_Contact(in1 := #Comp[1].Sts.RunSeconds, in2 := #MaxRunTime)
      wire#w1
      Move(in := #Comp[1].Sts.RunSeconds, out1 => #MaxRunTime)
   END_RUNG
   RUNG wire#w1
      Move(in := 1, out1 => #StopCandidate)
   END_RUNG
   // the same network as SCL:
   #_w1 := #Comp[1].Cmd.StartRequest AND (#Comp[1].Sts.RunSeconds > #MaxRunTime);
   IF #_w1 THEN
       #MaxRunTime := #Comp[1].Sts.RunSeconds;
       #StopCandidate := 1;
   END_IF;
END_REGION

REGION Network 41
   RUNG wire#powerrail
      Contact( #Comp[2].Cmd.StartRequest )
      { S7_Templates := "SrcType := DInt" } GT_Contact(in1 := #Comp[2].Sts.RunSeconds, in2 := #MaxRunTime)
      wire#w1
      Move(in := #Comp[2].Sts.RunSeconds, out1 => #MaxRunTime)
   END_RUNG
   RUNG wire#w1
      Move(in := 2, out1 => #StopCandidate)
   END_RUNG
   // the same network as SCL:
   #_w1 := #Comp[2].Cmd.StartRequest AND (#Comp[2].Sts.RunSeconds > #MaxRunTime);
   IF #_w1 THEN
       #MaxRunTime := #Comp[2].Sts.RunSeconds;
       #StopCandidate := 2;
   END_IF;
END_REGION

REGION Network 42
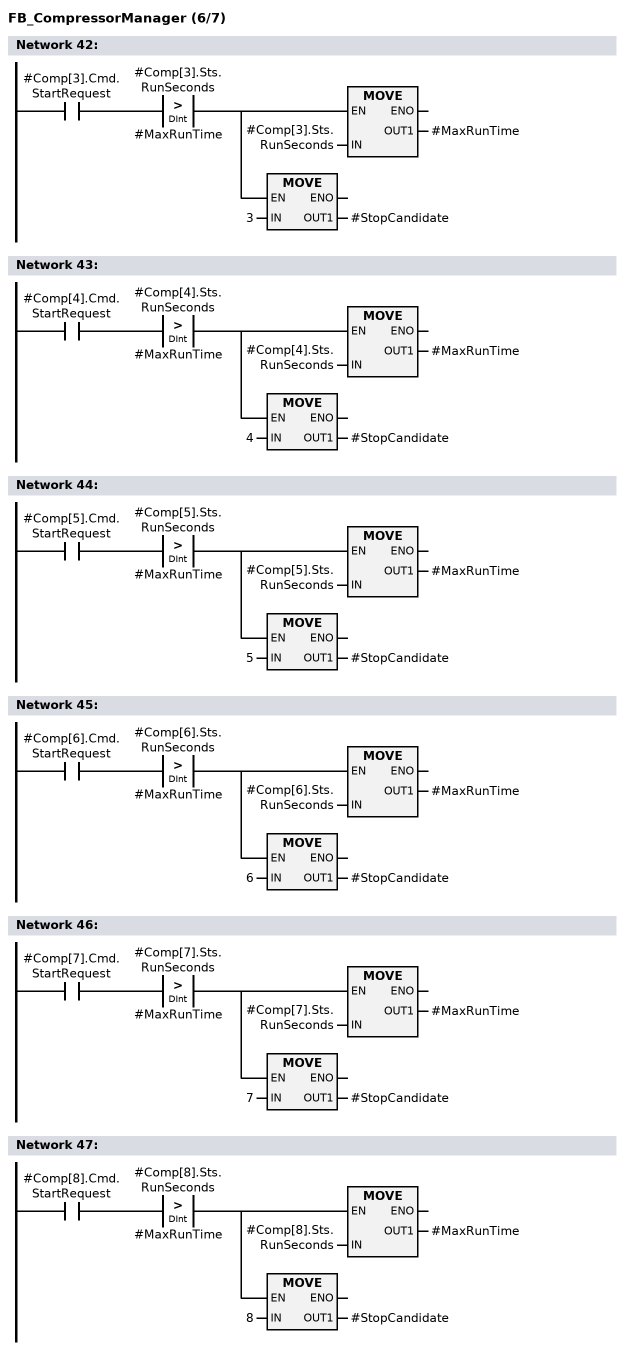
   RUNG wire#powerrail
      Contact( #Comp[3].Cmd.StartRequest )
      { S7_Templates := "SrcType := DInt" } GT_Contact(in1 := #Comp[3].Sts.RunSeconds, in2 := #MaxRunTime)
      wire#w1
      Move(in := #Comp[3].Sts.RunSeconds, out1 => #MaxRunTime)
   END_RUNG
   RUNG wire#w1
      Move(in := 3, out1 => #StopCandidate)
   END_RUNG
   // the same network as SCL:
   #_w1 := #Comp[3].Cmd.StartRequest AND (#Comp[3].Sts.RunSeconds > #MaxRunTime);
   IF #_w1 THEN
       #MaxRunTime := #Comp[3].Sts.RunSeconds;
       #StopCandidate := 3;
   END_IF;
END_REGION

REGION Network 43
   RUNG wire#powerrail
      Contact( #Comp[4].Cmd.StartRequest )
      { S7_Templates := "SrcType := DInt" } GT_Contact(in1 := #Comp[4].Sts.RunSeconds, in2 := #MaxRunTime)
      wire#w1
      Move(in := #Comp[4].Sts.RunSeconds, out1 => #MaxRunTime)
   END_RUNG
   RUNG wire#w1
      Move(in := 4, out1 => #StopCandidate)
   END_RUNG
   // the same network as SCL:
   #_w1 := #Comp[4].Cmd.StartRequest AND (#Comp[4].Sts.RunSeconds > #MaxRunTime);
   IF #_w1 THEN
       #MaxRunTime := #Comp[4].Sts.RunSeconds;
       #StopCandidate := 4;
   END_IF;
END_REGION

REGION Network 44
   RUNG wire#powerrail
      Contact( #Comp[5].Cmd.StartRequest )
      { S7_Templates := "SrcType := DInt" } GT_Contact(in1 := #Comp[5].Sts.RunSeconds, in2 := #MaxRunTime)
      wire#w1
      Move(in := #Comp[5].Sts.RunSeconds, out1 => #MaxRunTime)
   END_RUNG
   RUNG wire#w1
      Move(in := 5, out1 => #StopCandidate)
   END_RUNG
   // the same network as SCL:
   #_w1 := #Comp[5].Cmd.StartRequest AND (#Comp[5].Sts.RunSeconds > #MaxRunTime);
   IF #_w1 THEN
       #MaxRunTime := #Comp[5].Sts.RunSeconds;
       #StopCandidate := 5;
   END_IF;
END_REGION

REGION Network 45
   RUNG wire#powerrail
      Contact( #Comp[6].Cmd.StartRequest )
      { S7_Templates := "SrcType := DInt" } GT_Contact(in1 := #Comp[6].Sts.RunSeconds, in2 := #MaxRunTime)
      wire#w1
      Move(in := #Comp[6].Sts.RunSeconds, out1 => #MaxRunTime)
   END_RUNG
   RUNG wire#w1
      Move(in := 6, out1 => #StopCandidate)
   END_RUNG
   // the same network as SCL:
   #_w1 := #Comp[6].Cmd.StartRequest AND (#Comp[6].Sts.RunSeconds > #MaxRunTime);
   IF #_w1 THEN
       #MaxRunTime := #Comp[6].Sts.RunSeconds;
       #StopCandidate := 6;
   END_IF;
END_REGION

REGION Network 46
   RUNG wire#powerrail
      Contact( #Comp[7].Cmd.StartRequest )
      { S7_Templates := "SrcType := DInt" } GT_Contact(in1 := #Comp[7].Sts.RunSeconds, in2 := #MaxRunTime)
      wire#w1
      Move(in := #Comp[7].Sts.RunSeconds, out1 => #MaxRunTime)
   END_RUNG
   RUNG wire#w1
      Move(in := 7, out1 => #StopCandidate)
   END_RUNG
   // the same network as SCL:
   #_w1 := #Comp[7].Cmd.StartRequest AND (#Comp[7].Sts.RunSeconds > #MaxRunTime);
   IF #_w1 THEN
       #MaxRunTime := #Comp[7].Sts.RunSeconds;
       #StopCandidate := 7;
   END_IF;
END_REGION

REGION Network 47
   RUNG wire#powerrail
      Contact( #Comp[8].Cmd.StartRequest )
      { S7_Templates := "SrcType := DInt" } GT_Contact(in1 := #Comp[8].Sts.RunSeconds, in2 := #MaxRunTime)
      wire#w1
      Move(in := #Comp[8].Sts.RunSeconds, out1 => #MaxRunTime)
   END_RUNG
   RUNG wire#w1
      Move(in := 8, out1 => #StopCandidate)
   END_RUNG
   // the same network as SCL:
   #_w1 := #Comp[8].Cmd.StartRequest AND (#Comp[8].Sts.RunSeconds > #MaxRunTime);
   IF #_w1 THEN
       #MaxRunTime := #Comp[8].Sts.RunSeconds;
       #StopCandidate := 8;
   END_IF;
END_REGION

REGION Network 48
